LIN {X 0,Y 402.646,Z 650.506,A -85,B 0,C 180,E1 19904.527,E2 19904.527} C_VEL
LIN {X 0,Y 402.658,Z 650.513,A -85,B 0,C 180,E1 19900.591,E2 19900.591} C_VEL
LIN {X 0,Y 402.639,Z 650.511,A -85,B 0,C 180,E1 19896.705,E2 19896.705} C_VEL
LIN {X 0,Y 402.614,Z 650.499,A -85,B 0,C 180,E1 19892.849,E2 19892.849} C_VEL
LIN {X 0,Y 402.66,Z 650.51,A -85,B 0,C 180,E1 19889.006,E2 19889.006} C_VEL
LIN {X 0,Y 402.664,Z 650.497,A -85,B 0,C 180,E1 19885.016,E2 19885.016} C_VEL
LIN {X 0,Y 402.643,Z 650.508,A -85,B 0,C 180,E1 19881.145,E2 19881.145} C_VEL
LIN {X 0,Y 402.604,Z 650.504,A -85,B 0,C 180,E1 19877.232,E2 19877.232} C_VEL
LIN {X 0,Y 402.609,Z 650.515,A -85,B 0,C 180,E1 19873.259,E2 19873.259} C_VEL
LIN {X 0,Y 402.648,Z 650.51,A -85,B 0,C 180,E1 19869.354,E2 19869.354} C_VEL
LIN {X 0,Y 402.661,Z 650.512,A -85,B 0,C 180,E1 19865.502,E2 19865.502} C_VEL
LIN {X 0,Y 402.651,Z 650.512,A -85,B 0,C 180,E1 19861.689,E2 19861.689} C_VEL
LIN {X 0,Y 402.624,Z 650.516,A -85,B 0,C 180,E1 19857.863,E2 19857.863} C_VEL
LIN {X 0,Y 402.648,Z 650.514,A -85,B 0,C 180,E1 19853.95,E2 19853.95} C_VEL
LIN {X 0,Y 402.656,Z 650.511,A -85,B 0,C 180,E1 19851.843,E2 19851.843} C_VEL
LIN {X 0,Y 402.481,Z 651.272,A -85,B 0,C 180,E1 19851.242,E2 19851.242} C_VEL
LIN {X 0,Y 402.023,Z 653.793,A -85,B 0,C 180,E1 19850.558,E2 19850.558} C_VEL
LIN {X 0,Y 401.315,Z 659.057,A -85,B 0,C 180,E1 19849.745,E2 19849.745} C_VEL
LIN {X 0,Y 401.053,Z 668.633,A -85,B 0,C 180,E1 19848.719,E2 19848.719} C_VEL
LIN {X 0,Y 402.027,Z 674.176,A -85,B 0,C 180,E1 19848.104,E2 19848.104} C_VEL
LIN {X 0,Y 409.059,Z 698.473,A -85,B 0,C 180,E1 19845.257,E2 19845.257} C_VEL
LIN {X 0,Y 410.986,Z 706.413,A -85,B 0,C 180,E1 19844.378,E2 19844.378} C_VEL
LIN {X 0,Y 408.514,Z 749.372,A -85,B 0,C 180,E1 19840.433,E2 19840.433} C_VEL
LIN {X 0,Y 406.006,Z 793.704,A -85,B 0,C 180,E1 19836.364,E2 19836.364} C_VEL
LIN {X 0,Y 403.596,Z 838.675,A -85,B 0,C 180,E1 19832.264,E2 19832.264} C_VEL
LIN {X 0,Y 403.179,Z 847.022,A -85,B 0,C 180,E1 19831.548,E2 19831.548} C_VEL
LIN {X 0,Y 399.475,Z 984.558,A -85,B 0,C 180,E1 19828.359,E2 19828.359} C_VEL
LIN {X 0,Y 399.204,Z 1001.716,A -85,B 0,C 180,E1 19827.803,E2 19827.803} C_VEL
LIN {X 0,Y 398.675,Z 1018.522,A -85,B 0,C 180,E1 19826.993,E2 19826.993} C_VEL
LIN {X 0,Y 397.957,Z 1035.489,A -85,B 0,C 180,E1 19825.863,E2 19825.863} C_VEL
LIN {X 0,Y 397.14,Z 1050.63,A -85,B 0,C 180,E1 19824.542,E2 19824.542} C_VEL
LIN {X 0,Y 396.336,Z 1063.911,A -85,B 0,C 180,E1 19823.094,E2 19823.094} C_VEL
LIN {X 0,Y 395.475,Z 1077.222,A -85,B 0,C 180,E1 19821.269,E2 19821.269} C_VEL
LIN {X 0,Y 394.824,Z 1087.41,A -85,B 0,C 180,E1 19819.526,E2 19819.526} C_VEL
LIN {X 0,Y 394.308,Z 1096.659,A -85,B 0,C 180,E1 19817.558,E2 19817.558} C_VEL
LIN {X 0,Y 393.965,Z 1104.345,A -85,B 0,C 180,E1 19815.452,E2 19815.452} C_VEL
LIN {X 0,Y 393.819,Z 1110.47,A -85,B 0,C 180,E1 19813.206,E2 19813.206} C_VEL
LIN {X 0,Y 393.901,Z 1114.817,A -85,B 0,C 180,E1 19810.79,E2 19810.79} C_VEL
LIN {X 0,Y 394.207,Z 1116.994,A -85,B 0,C 180,E1 19808.603,E2 19808.603} C_VEL
LIN {X 0,Y 394.786,Z 1117.402,A -85,B 0,C 180,E1 19806.249,E2 19806.249} C_VEL
LIN {X 0,Y 395.615,Z 1116.078,A -85,B 0,C 180,E1 19804.055,E2 19804.055} C_VEL
LIN {X 0,Y 396.728,Z 1112.949,A -85,B 0,C 180,E1 19801.874,E2 19801.874} C_VEL
LIN {X 0,Y 398.17,Z 1108.026,A -85,B 0,C 180,E1 19799.709,E2 19799.709} C_VEL
LIN {X 0,Y 399.817,Z 1101.607,A -85,B 0,C 180,E1 19797.704,E2 19797.704} C_VEL
LIN {X 0,Y 401.766,Z 1093.191,A -85,B 0,C 180,E1 19795.715,E2 19795.715} C_VEL
LIN {X 0,Y 403.641,Z 1084.014,A -85,B 0,C 180,E1 19794.025,E2 19794.025} C_VEL
LIN {X 0,Y 405.893,Z 1071.581,A -85,B 0,C 180,E1 19792.21,E2 19792.21} C_VEL
LIN {X 0,Y 407.919,Z 1058.287,A -85,B 0,C 180,E1 19790.687,E2 19790.687} C_VEL
LIN {X 0,Y 409.629,Z 1044.619,A -85,B 0,C 180,E1 19789.448,E2 19789.448} C_VEL
LIN {X 0,Y 410.963,Z 1031.006,A -85,B 0,C 180,E1 19788.489,E2 19788.489} C_VEL
LIN {X 0,Y 411.947,Z 1018.129,A -85,B 0,C 180,E1 19787.771,E2 19787.771} C_VEL
LIN {X 0,Y 412.78,Z 1003.186,A -85,B 0,C 180,E1 19787.125,E2 19787.125} C_VEL
LIN {X 0,Y 414.292,Z 966.661,A -85,B 0,C 180,E1 19786.089,E2 19786.089} C_VEL
LIN {X 0,Y 421.684,Z 861.807,A -85,B 0,C 180,E1 19783.324,E2 19783.324} C_VEL
LIN {X 0,Y 426.377,Z 817.793,A -85,B 0,C 180,E1 19779.187,E2 19779.187} C_VEL
LIN {X 0,Y 431.826,Z 773.389,A -85,B 0,C 180,E1 19775,E2 19775} C_VEL
LIN {X 0,Y 437.615,Z 731.795,A -85,B 0,C 180,E1 19771.052,E2 19771.052} C_VEL
LIN {X 0,Y 435.458,Z 721.684,A -85,B 0,C 180,E1 19769.174,E2 19769.174} C_VEL
LIN {X 0,Y 432.981,Z 712.906,A -85,B 0,C 180,E1 19767.13,E2 19767.13} C_VEL
LIN {X 0,Y 430.66,Z 706.333,A -85,B 0,C 180,E1 19765.167,E2 19765.167} C_VEL
LIN {X 0,Y 429.171,Z 702.425,A -85,B 0,C 180,E1 19763.714,E2 19763.714} C_VEL
LIN {X 0,Y 427.98,Z 699.173,A -85,B 0,C 180,E1 19762.255,E2 19762.255} C_VEL
LIN {X 0,Y 426.868,Z 695.743,A -85,B 0,C 180,E1 19760.198,E2 19760.198} C_VEL
LIN {X 0,Y 426.506,Z 695.015,A -85,B 0,C 180,E1 19759.423,E2 19759.423} C_VEL
LIN {X 0,Y 426.307,Z 694.895,A -85,B 0,C 180,E1 19759.043,E2 19759.043} C_VEL
LIN {X 0,Y 424.791,Z 697.509,A -85,B 0,C 180,E1 19758.047,E2 19758.047} C_VEL
LIN {X 0,Y 423.827,Z 699.741,A -85,B 0,C 180,E1 19757.294,E2 19757.294} C_VEL
LIN {X 0,Y 420.94,Z 708.266,A -85,B 0,C 180,E1 19755.654,E2 19755.654} C_VEL
LIN {X 0,Y 437.029,Z 740.937,A -85,B 0,C 180,E1 19753.195,E2 19753.195} C_VEL
LIN {X 0,Y 439.901,Z 747.523,A -85,B 0,C 180,E1 19752.76,E2 19752.76} C_VEL
LIN {X 0,Y 425.069,Z 979.024,A -85,B 0,C 180,E1 19747.665,E2 19747.665} C_VEL
LIN {X 0,Y 422.711,Z 1003.261,A -85,B 0,C 180,E1 19746.883,E2 19746.883} C_VEL
LIN {X 0,Y 419.964,Z 1026.175,A -85,B 0,C 180,E1 19745.884,E2 19745.884} C_VEL
LIN {X 0,Y 417.024,Z 1047.578,A -85,B 0,C 180,E1 19744.7,E2 19744.7} C_VEL
LIN {X 0,Y 413.637,Z 1069.6,A -85,B 0,C 180,E1 19743.201,E2 19743.201} C_VEL
LIN {X 0,Y 410.261,Z 1089.995,A -85,B 0,C 180,E1 19741.516,E2 19741.516} C_VEL
LIN {X 0,Y 406.993,Z 1108.788,A -85,B 0,C 180,E1 19739.67,E2 19739.67} C_VEL
LIN {X 0,Y 403.746,Z 1126.909,A -85,B 0,C 180,E1 19737.547,E2 19737.547} C_VEL
LIN {X 0,Y 400.86,Z 1142.981,A -85,B 0,C 180,E1 19735.324,E2 19735.324} C_VEL
LIN {X 0,Y 398.15,Z 1158.777,A -85,B 0,C 180,E1 19732.75,E2 19732.75} C_VEL
LIN {X 0,Y 396.073,Z 1171.861,A -85,B 0,C 180,E1 19730.232,E2 19730.232} C_VEL
LIN {X 0,Y 394.432,Z 1183.554,A -85,B 0,C 180,E1 19727.555,E2 19727.555} C_VEL
LIN {X 0,Y 393.294,Z 1193.275,A -85,B 0,C 180,E1 19724.877,E2 19724.877} C_VEL
LIN {X 0,Y 392.561,Z 1201.854,A -85,B 0,C 180,E1 19722.009,E2 19722.009} C_VEL
LIN {X 0,Y 392.233,Z 1208.397,A -85,B 0,C 180,E1 19719.24,E2 19719.24} C_VEL
LIN {X 0,Y 392.151,Z 1213.369,A -85,B 0,C 180,E1 19716.439,E2 19716.439} C_VEL
LIN {X 0,Y 392.187,Z 1216.843,A -85,B 0,C 180,E1 19713.652,E2 19713.652} C_VEL
LIN {X 0,Y 392.216,Z 1218.667,A -85,B 0,C 180,E1 19710.874,E2 19710.874} C_VEL
LIN {X 0,Y 392.161,Z 1219.127,A -85,B 0,C 180,E1 19708.099,E2 19708.099} C_VEL
LIN {X 0,Y 392.064,Z 1217.981,A -85,B 0,C 180,E1 19705.317,E2 19705.317} C_VEL
LIN {X 0,Y 392.055,Z 1215.324,A -85,B 0,C 180,E1 19702.377,E2 19702.377} C_VEL
LIN {X 0,Y 392.305,Z 1211.002,A -85,B 0,C 180,E1 19699.424,E2 19699.424} C_VEL
LIN {X 0,Y 393.041,Z 1204.73,A -85,B 0,C 180,E1 19696.313,E2 19696.313} C_VEL
LIN {X 0,Y 394.347,Z 1197.092,A -85,B 0,C 180,E1 19693.349,E2 19693.349} C_VEL
LIN {X 0,Y 396.474,Z 1187.039,A -85,B 0,C 180,E1 19690.247,E2 19690.247} C_VEL
LIN {X 0,Y 399.332,Z 1175.533,A -85,B 0,C 180,E1 19687.317,E2 19687.317} C_VEL
LIN {X 0,Y 403.067,Z 1161.949,A -85,B 0,C 180,E1 19684.427,E2 19684.427} C_VEL
LIN {X 0,Y 407.523,Z 1146.959,A -85,B 0,C 180,E1 19681.734,E2 19681.734} C_VEL
LIN {X 0,Y 413.055,Z 1129.099,A -85,B 0,C 180,E1 19679.041,E2 19679.041} C_VEL
LIN {X 0,Y 419.266,Z 1109.523,A -85,B 0,C 180,E1 19676.569,E2 19676.569} C_VEL
LIN {X 0,Y 425.881,Z 1088.959,A -85,B 0,C 180,E1 19674.389,E2 19674.389} C_VEL
LIN {X 0,Y 433,Z 1066.974,A -85,B 0,C 180,E1 19672.436,E2 19672.436} C_VEL
LIN {X 0,Y 440.578,Z 1043.466,A -85,B 0,C 180,E1 19670.713,E2 19670.713} C_VEL
LIN {X 0,Y 448.214,Z 1019.183,A -85,B 0,C 180,E1 19669.267,E2 19669.267} C_VEL
LIN {X 0,Y 455.498,Z 995.065,A -85,B 0,C 180,E1 19668.137,E2 19668.137} C_VEL
LIN {X 0,Y 462.97,Z 967.876,A -85,B 0,C 180,E1 19667.141,E2 19667.141} C_VEL
LIN {X 0,Y 483.825,Z 882.658,A -85,B 0,C 180,E1 19664.617,E2 19664.617} C_VEL
LIN {X 0,Y 466.018,Z 953.723,A -85,B 0,C 180,E1 19662.524,E2 19662.524} C_VEL
LIN {X 0,Y 459.927,Z 976.756,A -85,B 0,C 180,E1 19661.621,E2 19661.621} C_VEL
LIN {X 0,Y 453.131,Z 999.954,A -85,B 0,C 180,E1 19660.45,E2 19660.45} C_VEL
LIN {X 0,Y 446.12,Z 1022.308,A -85,B 0,C 180,E1 19659.038,E2 19659.038} C_VEL
LIN {X 0,Y 438.753,Z 1044.675,A -85,B 0,C 180,E1 19657.31,E2 19657.31} C_VEL
LIN {X 0,Y 431.735,Z 1065.276,A -85,B 0,C 180,E1 19655.383,E2 19655.383} C_VEL
LIN {X 0,Y 425.061,Z 1084.433,A -85,B 0,C 180,E1 19653.239,E2 19653.239} C_VEL
LIN {X 0,Y 418.789,Z 1102.064,A -85,B 0,C 180,E1 19650.889,E2 19650.889} C_VEL
LIN {X 0,Y 413.031,Z 1118.126,A -85,B 0,C 180,E1 19648.329,E2 19648.329} C_VEL
LIN {X 0,Y 408.086,Z 1131.941,A -85,B 0,C 180,E1 19645.704,E2 19645.704} C_VEL
LIN {X 0,Y 403.945,Z 1143.775,A -85,B 0,C 180,E1 19643.026,E2 19643.026} C_VEL
LIN {X 0,Y 400.198,Z 1154.642,A -85,B 0,C 180,E1 19640.019,E2 19640.019} C_VEL
LIN {X 0,Y 397.338,Z 1163.443,A -85,B 0,C 180,E1 19637.005,E2 19637.005} C_VEL
LIN {X 0,Y 395.122,Z 1170.858,A -85,B 0,C 180,E1 19633.764,E2 19633.764} C_VEL
LIN {X 0,Y 393.737,Z 1176.111,A -85,B 0,C 180,E1 19630.686,E2 19630.686} C_VEL
LIN {X 0,Y 392.874,Z 1179.647,A -85,B 0,C 180,E1 19627.608,E2 19627.608} C_VEL
LIN {X 0,Y 392.42,Z 1181.535,A -85,B 0,C 180,E1 19624.533,E2 19624.533} C_VEL
LIN {X 0,Y 392.235,Z 1181.899,A -85,B 0,C 180,E1 19621.61,E2 19621.61} C_VEL
LIN {X 0,Y 392.162,Z 1180.769,A -85,B 0,C 180,E1 19618.834,E2 19618.834} C_VEL
LIN {X 0,Y 392.176,Z 1177.983,A -85,B 0,C 180,E1 19615.763,E2 19615.763} C_VEL
LIN {X 0,Y 392.357,Z 1173.769,A -85,B 0,C 180,E1 19612.83,E2 19612.83} C_VEL
LIN {X 0,Y 392.769,Z 1167.777,A -85,B 0,C 180,E1 19609.887,E2 19609.887} C_VEL
LIN {X 0,Y 393.54,Z 1160.062,A -85,B 0,C 180,E1 19606.934,E2 19606.934} C_VEL
LIN {X 0,Y 394.697,Z 1150.979,A -85,B 0,C 180,E1 19604.125,E2 19604.125} C_VEL
LIN {X 0,Y 396.355,Z 1139.874,A -85,B 0,C 180,E1 19601.318,E2 19601.318} C_VEL
LIN {X 0,Y 398.437,Z 1127.317,A -85,B 0,C 180,E1 19598.665,E2 19598.665} C_VEL
LIN {X 0,Y 401.054,Z 1112.484,A -85,B 0,C 180,E1 19596.026,E2 19596.026} C_VEL
LIN {X 0,Y 403.937,Z 1096.683,A -85,B 0,C 180,E1 19593.65,E2 19593.65} C_VEL
LIN {X 0,Y 407.051,Z 1079.568,A -85,B 0,C 180,E1 19591.464,E2 19591.464} C_VEL
LIN {X 0,Y 410.306,Z 1060.961,A -85,B 0,C 180,E1 19589.467,E2 19589.467} C_VEL
LIN {X 0,Y 413.532,Z 1041.496,A -85,B 0,C 180,E1 19587.704,E2 19587.704} C_VEL
LIN {X 0,Y 416.755,Z 1020.503,A -85,B 0,C 180,E1 19586.114,E2 19586.114} C_VEL
LIN {X 0,Y 419.661,Z 999.367,A -85,B 0,C 180,E1 19584.793,E2 19584.793} C_VEL
LIN {X 0,Y 422.338,Z 977.144,A -85,B 0,C 180,E1 19583.672,E2 19583.672} C_VEL
LIN {X 0,Y 424.639,Z 953.609,A -85,B 0,C 180,E1 19582.759,E2 19582.759} C_VEL
LIN {X 0,Y 426.356,Z 930.684,A -85,B 0,C 180,E1 19582.109,E2 19582.109} C_VEL
LIN {X 0,Y 438.997,Z 728.954,A -85,B 0,C 180,E1 19577.705,E2 19577.705} C_VEL
LIN {X 0,Y 420.147,Z 695.163,A -85,B 0,C 180,E1 19574.978,E2 19574.978} C_VEL
LIN {X 0,Y 403.964,Z 667.893,A -85,B 0,C 180,E1 19572.44,E2 19572.44} C_VEL
LIN {X 0,Y 396.718,Z 655.938,A -85,B 0,C 180,E1 19571.232,E2 19571.232} C_VEL
LIN {X 0,Y 394.919,Z 652.752,A -85,B 0,C 180,E1 19570.918,E2 19570.918} C_VEL
LIN {X 0,Y 394.665,Z 651.506,A -85,B 0,C 180,E1 19570.819,E2 19570.819} C_VEL
LIN {X 0,Y 394.674,Z 651.506,A -85,B 0,C 180,E1 19566.822,E2 19566.822} C_VEL
LIN {X 0,Y 394.713,Z 651.496,A -85,B 0,C 180,E1 19562.829,E2 19562.829} C_VEL
LIN {X 0,Y 394.726,Z 651.495,A -85,B 0,C 180,E1 19558.937,E2 19558.937} C_VEL
LIN {X 0,Y 394.696,Z 651.503,A -85,B 0,C 180,E1 19555.03,E2 19555.03} C_VEL
LIN {X 0,Y 394.665,Z 651.508,A -85,B 0,C 180,E1 19551.087,E2 19551.087} C_VEL
LIN {X 0,Y 394.702,Z 651.497,A -85,B 0,C 180,E1 19547.243,E2 19547.243} C_VEL
LIN {X 0,Y 394.727,Z 651.485,A -85,B 0,C 180,E1 19543.329,E2 19543.329} C_VEL
LIN {X 0,Y 394.719,Z 651.492,A -85,B 0,C 180,E1 19539.332,E2 19539.332} C_VEL
LIN {X 0,Y 394.688,Z 651.505,A -85,B 0,C 180,E1 19535.415,E2 19535.415} C_VEL
LIN {X 0,Y 394.694,Z 651.492,A -85,B 0,C 180,E1 19531.308,E2 19531.308} C_VEL
LIN {X 0,Y 394.72,Z 651.487,A -85,B 0,C 180,E1 19527.389,E2 19527.389} C_VEL
LIN {X 0,Y 394.715,Z 651.5,A -85,B 0,C 180,E1 19523.457,E2 19523.457} C_VEL
LIN {X 0,Y 394.682,Z 651.483,A -85,B 0,C 180,E1 19519.492,E2 19519.492} C_VEL
LIN {X 0,Y 394.649,Z 651.506,A -85,B 0,C 180,E1 19515.476,E2 19515.476} C_VEL
LIN {X 0,Y 394.684,Z 651.503,A -85,B 0,C 180,E1 19511.541,E2 19511.541} C_VEL
LIN {X 0,Y 394.717,Z 651.502,A -85,B 0,C 180,E1 19507.599,E2 19507.599} C_VEL
LIN {X 0,Y 394.724,Z 651.498,A -85,B 0,C 180,E1 19503.688,E2 19503.688} C_VEL
LIN {X 0,Y 394.692,Z 651.504,A -85,B 0,C 180,E1 19499.745,E2 19499.745} C_VEL
LIN {X 0,Y 394.687,Z 651.506,A -85,B 0,C 180,E1 19495.781,E2 19495.781} C_VEL
LIN {X 0,Y 394.717,Z 651.5,A -85,B 0,C 180,E1 19491.826,E2 19491.826} C_VEL
LIN {X 0,Y 394.735,Z 651.678,A -85,B 0,C 180,E1 19490.866,E2 19490.866} C_VEL
LIN {X 0,Y 402.027,Z 674.176,A -85,B 0,C 180,E1 19488.104,E2 19488.104} C_VEL
LIN {X 0,Y 402.871,Z 680.333,A -85,B 0,C 180,E1 19487.442,E2 19487.442} C_VEL
LIN {X 0,Y 401.632,Z 699.052,A -85,B 0,C 180,E1 19485.691,E2 19485.691} C_VEL
LIN {X 0,Y 402.317,Z 703.478,A -85,B 0,C 180,E1 19485.217,E2 19485.217} C_VEL
LIN {X 0,Y 403.454,Z 708.427,A -85,B 0,C 180,E1 19484.665,E2 19484.665} C_VEL
LIN {X 0,Y 400.84,Z 752.044,A -85,B 0,C 180,E1 19480.616,E2 19480.616} C_VEL
LIN {X 0,Y 398.274,Z 796.537,A -85,B 0,C 180,E1 19476.508,E2 19476.508} C_VEL
LIN {X 0,Y 395.755,Z 842.489,A -85,B 0,C 180,E1 19472.272,E2 19472.272} C_VEL
LIN {X 0,Y 395.417,Z 847.822,A -85,B 0,C 180,E1 19471.823,E2 19471.823} C_VEL
LIN {X 0,Y 391.587,Z 985.022,A -85,B 0,C 180,E1 19468.547,E2 19468.547} C_VEL
LIN {X 0,Y 391.307,Z 1002.317,A -85,B 0,C 180,E1 19467.979,E2 19467.979} C_VEL
LIN {X 0,Y 390.777,Z 1018.864,A -85,B 0,C 180,E1 19467.172,E2 19467.172} C_VEL
LIN {X 0,Y 390.074,Z 1035.219,A -85,B 0,C 180,E1 19466.075,E2 19466.075} C_VEL
LIN {X 0,Y 389.296,Z 1049.667,A -85,B 0,C 180,E1 19464.827,E2 19464.827} C_VEL
LIN {X 0,Y 388.394,Z 1064.416,A -85,B 0,C 180,E1 19463.217,E2 19463.217} C_VEL
LIN {X 0,Y 387.569,Z 1076.966,A -85,B 0,C 180,E1 19461.487,E2 19461.487} C_VEL
LIN {X 0,Y 386.868,Z 1087.854,A -85,B 0,C 180,E1 19459.629,E2 19459.629} C_VEL
LIN {X 0,Y 386.309,Z 1097.863,A -85,B 0,C 180,E1 19457.469,E2 19457.469} C_VEL
LIN {X 0,Y 385.974,Z 1105.522,A -85,B 0,C 180,E1 19455.318,E2 19455.318} C_VEL
LIN {X 0,Y 385.846,Z 1111.603,A -85,B 0,C 180,E1 19453.026,E2 19453.026} C_VEL
LIN {X 0,Y 385.959,Z 1115.863,A -85,B 0,C 180,E1 19450.596,E2 19450.596} C_VEL
LIN {X 0,Y 386.312,Z 1118.066,A -85,B 0,C 180,E1 19448.331,E2 19448.331} C_VEL
LIN {X 0,Y 386.959,Z 1118.458,A -85,B 0,C 180,E1 19445.929,E2 19445.929} C_VEL
LIN {X 0,Y 387.871,Z 1117.094,A -85,B 0,C 180,E1 19443.692,E2 19443.692} C_VEL
LIN {X 0,Y 389.181,Z 1113.683,A -85,B 0,C 180,E1 19441.322,E2 19441.322} C_VEL
LIN {X 0,Y 390.768,Z 1108.625,A -85,B 0,C 180,E1 19439.117,E2 19439.117} C_VEL
LIN {X 0,Y 392.704,Z 1101.473,A -85,B 0,C 180,E1 19436.932,E2 19436.932} C_VEL
LIN {X 0,Y 394.668,Z 1093.37,A -85,B 0,C 180,E1 19435.055,E2 19435.055} C_VEL
LIN {X 0,Y 396.877,Z 1083.175,A -85,B 0,C 180,E1 19433.197,E2 19433.197} C_VEL
LIN {X 0,Y 399.022,Z 1071.886,A -85,B 0,C 180,E1 19431.568,E2 19431.568} C_VEL
LIN {X 0,Y 401.176,Z 1058.387,A -85,B 0,C 180,E1 19430.022,E2 19430.022} C_VEL
LIN {X 0,Y 403.1,Z 1043.582,A -85,B 0,C 180,E1 19428.696,E2 19428.696} C_VEL
LIN {X 0,Y 404.436,Z 1030.633,A -85,B 0,C 180,E1 19427.794,E2 19427.794} C_VEL
LIN {X 0,Y 405.446,Z 1018.234,A -85,B 0,C 180,E1 19427.101,E2 19427.101} C_VEL
LIN {X 0,Y 406.28,Z 1003.609,A -85,B 0,C 180,E1 19426.472,E2 19426.472} C_VEL
LIN {X 0,Y 408.076,Z 964.911,A -85,B 0,C 180,E1 19425.356,E2 19425.356} C_VEL
LIN {X 0,Y 415.65,Z 863.65,A -85,B 0,C 180,E1 19422.642,E2 19422.642} C_VEL
LIN {X 0,Y 420.636,Z 820.445,A -85,B 0,C 180,E1 19418.524,E2 19418.524} C_VEL
LIN {X 0,Y 426.779,Z 774.226,A -85,B 0,C 180,E1 19414.108,E2 19414.108} C_VEL
LIN {X 0,Y 432.533,Z 736.055,A -85,B 0,C 180,E1 19410.416,E2 19410.416} C_VEL
LIN {X 0,Y 430.698,Z 726.646,A -85,B 0,C 180,E1 19408.585,E2 19408.585} C_VEL
LIN {X 0,Y 428.479,Z 718.439,A -85,B 0,C 180,E1 19406.581,E2 19406.581} C_VEL
LIN {X 0,Y 426.54,Z 712.406,A -85,B 0,C 180,E1 19404.66,E2 19404.66} C_VEL
LIN {X 0,Y 425.512,Z 709.318,A -85,B 0,C 180,E1 19403.475,E2 19403.475} C_VEL
LIN {X 0,Y 424.538,Z 706.275,A -85,B 0,C 180,E1 19402.066,E2 19402.066} C_VEL
LIN {X 0,Y 423.625,Z 703.028,A -85,B 0,C 180,E1 19400.056,E2 19400.056} C_VEL
LIN {X 0,Y 423.337,Z 702.308,A -85,B 0,C 180,E1 19399.248,E2 19399.248} C_VEL
LIN {X 0,Y 421.274,Z 706.106,A -85,B 0,C 180,E1 19397.874,E2 19397.874} C_VEL
LIN {X 0,Y 417.335,Z 717.08,A -85,B 0,C 180,E1 19395.741,E2 19395.741} C_VEL
LIN {X 0,Y 433.11,Z 749.566,A -85,B 0,C 180,E1 19393.301,E2 19393.301} C_VEL
LIN {X 0,Y 417.912,Z 978.657,A -85,B 0,C 180,E1 19388.153,E2 19388.153} C_VEL
LIN {X 0,Y 415.516,Z 1002.68,A -85,B 0,C 180,E1 19387.364,E2 19387.364} C_VEL
LIN {X 0,Y 412.727,Z 1025.325,A -85,B 0,C 180,E1 19386.363,E2 19386.363} C_VEL
LIN {X 0,Y 409.688,Z 1046.975,A -85,B 0,C 180,E1 19385.151,E2 19385.151} C_VEL
LIN {X 0,Y 406.211,Z 1069.033,A -85,B 0,C 180,E1 19383.628,E2 19383.628} C_VEL
LIN {X 0,Y 402.754,Z 1089.393,A -85,B 0,C 180,E1 19381.922,E2 19381.922} C_VEL
LIN {X 0,Y 399.402,Z 1108.229,A -85,B 0,C 180,E1 19380.043,E2 19380.043} C_VEL
LIN {X 0,Y 396.006,Z 1126.687,A -85,B 0,C 180,E1 19377.844,E2 19377.844} C_VEL
LIN {X 0,Y 393.005,Z 1142.992,A -85,B 0,C 180,E1 19375.544,E2 19375.544} C_VEL
LIN {X 0,Y 390.378,Z 1157.917,A -85,B 0,C 180,E1 19373.069,E2 19373.069} C_VEL
LIN {X 0,Y 388.226,Z 1171.099,A -85,B 0,C 180,E1 19370.501,E2 19370.501} C_VEL
LIN {X 0,Y 386.523,Z 1182.843,A -85,B 0,C 180,E1 19367.771,E2 19367.771} C_VEL
LIN {X 0,Y 385.344,Z 1192.641,A -85,B 0,C 180,E1 19365.037,E2 19365.037} C_VEL
LIN {X 0,Y 384.594,Z 1201.167,A -85,B 0,C 180,E1 19362.155,E2 19362.155} C_VEL
LIN {X 0,Y 384.249,Z 1207.849,A -85,B 0,C 180,E1 19359.282,E2 19359.282} C_VEL
LIN {X 0,Y 384.168,Z 1212.862,A -85,B 0,C 180,E1 19356.424,E2 19356.424} C_VEL
LIN {X 0,Y 384.206,Z 1216.352,A -85,B 0,C 180,E1 19353.579,E2 19353.579} C_VEL
LIN {X 0,Y 384.231,Z 1218.201,A -85,B 0,C 180,E1 19350.743,E2 19350.743} C_VEL
LIN {X 0,Y 384.167,Z 1218.671,A -85,B 0,C 180,E1 19347.91,E2 19347.91} C_VEL
LIN {X 0,Y 384.061,Z 1217.536,A -85,B 0,C 180,E1 19345.069,E2 19345.069} C_VEL
LIN {X 0,Y 384.063,Z 1214.9,A -85,B 0,C 180,E1 19342.067,E2 19342.067} C_VEL
LIN {X 0,Y 384.366,Z 1210.584,A -85,B 0,C 180,E1 19339.051,E2 19339.051} C_VEL
LIN {X 0,Y 385.255,Z 1204.012,A -85,B 0,C 180,E1 19335.724,E2 19335.724} C_VEL
LIN {X 0,Y 386.824,Z 1195.882,A -85,B 0,C 180,E1 19332.55,E2 19332.55} C_VEL
LIN {X 0,Y 389.23,Z 1185.771,A -85,B 0,C 180,E1 19329.392,E2 19329.392} C_VEL
LIN {X 0,Y 392.405,Z 1174.164,A -85,B 0,C 180,E1 19326.417,E2 19326.417} C_VEL
LIN {X 0,Y 396.748,Z 1159.803,A -85,B 0,C 180,E1 19323.345,E2 19323.345} C_VEL
LIN {X 0,Y 401.919,Z 1143.803,A -85,B 0,C 180,E1 19320.488,E2 19320.488} C_VEL
LIN {X 0,Y 407.83,Z 1126.286,A -85,B 0,C 180,E1 19317.856,E2 19317.856} C_VEL
LIN {X 0,Y 414.605,Z 1106.761,A -85,B 0,C 180,E1 19315.391,E2 19315.391} C_VEL
LIN {X 0,Y 421.996,Z 1085.741,A -85,B 0,C 180,E1 19313.167,E2 19313.167} C_VEL
LIN {X 0,Y 429.966,Z 1063.264,A -85,B 0,C 180,E1 19311.19,E2 19311.19} C_VEL
LIN {X 0,Y 438.413,Z 1039.238,A -85,B 0,C 180,E1 19309.457,E2 19309.457} C_VEL
LIN {X 0,Y 446.678,Z 1015.23,A -85,B 0,C 180,E1 19308.071,E2 19308.071} C_VEL
LIN {X 0,Y 454.455,Z 991.415,A -85,B 0,C 180,E1 19306.994,E2 19306.994} C_VEL
LIN {X 0,Y 462.394,Z 964.567,A -85,B 0,C 180,E1 19306.04,E2 19306.04} C_VEL
LIN {X 0,Y 474.662,Z 916.991,A -85,B 0,C 180,E1 19304.622,E2 19304.622} C_VEL
LIN {X 0,Y 463.429,Z 959.702,A -85,B 0,C 180,E1 19303.326,E2 19303.326} C_VEL
LIN {X 0,Y 456.454,Z 983.213,A -85,B 0,C 180,E1 19302.348,E2 19302.348} C_VEL
LIN {X 0,Y 448.781,Z 1006.559,A -85,B 0,C 180,E1 19301.094,E2 19301.094} C_VEL
LIN {X 0,Y 440.915,Z 1028.975,A -85,B 0,C 180,E1 19299.589,E2 19299.589} C_VEL
LIN {X 0,Y 433.026,Z 1050.608,A -85,B 0,C 180,E1 19297.814,E2 19297.814} C_VEL
LIN {X 0,Y 425.278,Z 1071.277,A -85,B 0,C 180,E1 19295.753,E2 19295.753} C_VEL
LIN {X 0,Y 418.168,Z 1089.948,A -85,B 0,C 180,E1 19293.531,E2 19293.531} C_VEL
LIN {X 0,Y 411.364,Z 1107.559,A -85,B 0,C 180,E1 19291.02,E2 19291.02} C_VEL
LIN {X 0,Y 405.16,Z 1123.521,A -85,B 0,C 180,E1 19288.286,E2 19288.286} C_VEL
LIN {X 0,Y 399.882,Z 1137.117,A -85,B 0,C 180,E1 19285.475,E2 19285.475} C_VEL
LIN {X 0,Y 395.49,Z 1148.605,A -85,B 0,C 180,E1 19282.603,E2 19282.603} C_VEL
LIN {X 0,Y 391.798,Z 1158.672,A -85,B 0,C 180,E1 19279.534,E2 19279.534} C_VEL
LIN {X 0,Y 388.975,Z 1166.853,A -85,B 0,C 180,E1 19276.428,E2 19276.428} C_VEL
LIN {X 0,Y 386.955,Z 1173.258,A -85,B 0,C 180,E1 19273.299,E2 19273.299} C_VEL
LIN {X 0,Y 385.591,Z 1177.858,A -85,B 0,C 180,E1 19270.159,E2 19270.159} C_VEL
LIN {X 0,Y 384.765,Z 1180.975,A -85,B 0,C 180,E1 19266.869,E2 19266.869} C_VEL
LIN {X 0,Y 384.386,Z 1182.339,A -85,B 0,C 180,E1 19263.881,E2 19263.881} C_VEL
LIN {X 0,Y 384.217,Z 1182.094,A -85,B 0,C 180,E1 19260.898,E2 19260.898} C_VEL
LIN {X 0,Y 384.155,Z 1180.301,A -85,B 0,C 180,E1 19257.766,E2 19257.766} C_VEL
LIN {X 0,Y 384.219,Z 1177.239,A -85,B 0,C 180,E1 19254.927,E2 19254.927} C_VEL
LIN {X 0,Y 384.456,Z 1172.39,A -85,B 0,C 180,E1 19251.93,E2 19251.93} C_VEL
LIN {X 0,Y 384.981,Z 1165.902,A -85,B 0,C 180,E1 19248.923,E2 19248.923} C_VEL
LIN {X 0,Y 385.905,Z 1157.583,A -85,B 0,C 180,E1 19245.907,E2 19245.907} C_VEL
LIN {X 0,Y 387.256,Z 1147.73,A -85,B 0,C 180,E1 19243.04,E2 19243.04} C_VEL
LIN {X 0,Y 389.145,Z 1135.888,A -85,B 0,C 180,E1 19240.178,E2 19240.178} C_VEL
LIN {X 0,Y 391.34,Z 1123.384,A -85,B 0,C 180,E1 19237.627,E2 19237.627} C_VEL
LIN {X 0,Y 394.043,Z 1108.674,A -85,B 0,C 180,E1 19235.092,E2 19235.092} C_VEL
LIN {X 0,Y 397.025,Z 1092.604,A -85,B 0,C 180,E1 19232.752,E2 19232.752} C_VEL
LIN {X 0,Y 400.345,Z 1074.618,A -85,B 0,C 180,E1 19230.531,E2 19230.531} C_VEL
LIN {X 0,Y 403.803,Z 1055.148,A -85,B 0,C 180,E1 19228.506,E2 19228.506} C_VEL
LIN {X 0,Y 407.073,Z 1035.559,A -85,B 0,C 180,E1 19226.791,E2 19226.791} C_VEL
LIN {X 0,Y 410.344,Z 1014.252,A -85,B 0,C 180,E1 19225.241,E2 19225.241} C_VEL
LIN {X 0,Y 413.297,Z 992.366,A -85,B 0,C 180,E1 19223.95,E2 19223.95} C_VEL
LIN {X 0,Y 415.883,Z 969.815,A -85,B 0,C 180,E1 19222.886,E2 19222.886} C_VEL
LIN {X 0,Y 418.114,Z 945.816,A -85,B 0,C 180,E1 19222.022,E2 19222.022} C_VEL
LIN {X 0,Y 420.091,Z 917.398,A -85,B 0,C 180,E1 19221.306,E2 19221.306} C_VEL
LIN {X 0,Y 432.144,Z 731.726,A -85,B 0,C 180,E1 19217.18,E2 19217.18} C_VEL
LIN {X 0,Y 413.501,Z 698.183,A -85,B 0,C 180,E1 19214.408,E2 19214.408} C_VEL
LIN {X 0,Y 396.406,Z 669.438,A -85,B 0,C 180,E1 19211.657,E2 19211.657} C_VEL
LIN {X 0,Y 389.378,Z 657.671,A -85,B 0,C 180,E1 19210.447,E2 19210.447} C_VEL
LIN {X 0,Y 387.126,Z 654.072,A -85,B 0,C 180,E1 19210.052,E2 19210.052} C_VEL
LIN {X 0,Y 386.751,Z 652.489,A -85,B 0,C 180,E1 19209.933,E2 19209.933} C_VEL
LIN {X 0,Y 386.77,Z 652.487,A -85,B 0,C 180,E1 19205.935,E2 19205.935} C_VEL
LIN {X 0,Y 386.789,Z 652.483,A -85,B 0,C 180,E1 19202.004,E2 19202.004} C_VEL
LIN {X 0,Y 386.779,Z 652.493,A -85,B 0,C 180,E1 19198.069,E2 19198.069} C_VEL
LIN {X 0,Y 386.746,Z 652.497,A -85,B 0,C 180,E1 19194.112,E2 19194.112} C_VEL
LIN {X 0,Y 386.73,Z 652.499,A -85,B 0,C 180,E1 19190.115,E2 19190.115} C_VEL
LIN {X 0,Y 386.768,Z 652.491,A -85,B 0,C 180,E1 19186.215,E2 19186.215} C_VEL
LIN {X 0,Y 386.781,Z 652.483,A -85,B 0,C 180,E1 19182.24,E2 19182.24} C_VEL
LIN {X 0,Y 386.751,Z 652.478,A -85,B 0,C 180,E1 19178.177,E2 19178.177} C_VEL
LIN {X 0,Y 386.712,Z 652.492,A -85,B 0,C 180,E1 19174.154,E2 19174.154} C_VEL
LIN {X 0,Y 386.737,Z 652.492,A -85,B 0,C 180,E1 19170.002,E2 19170.002} C_VEL
LIN {X 0,Y 386.771,Z 652.468,A -85,B 0,C 180,E1 19166,E2 19166} C_VEL
LIN {X 0,Y 386.78,Z 652.489,A -85,B 0,C 180,E1 19161.978,E2 19161.978} C_VEL
LIN {X 0,Y 386.742,Z 652.47,A -85,B 0,C 180,E1 19158.065,E2 19158.065} C_VEL
LIN {X 0,Y 386.732,Z 652.492,A -85,B 0,C 180,E1 19154.096,E2 19154.096} C_VEL
LIN {X 0,Y 386.77,Z 652.486,A -85,B 0,C 180,E1 19150.207,E2 19150.207} C_VEL
LIN {X 0,Y 386.789,Z 652.484,A -85,B 0,C 180,E1 19146.213,E2 19146.213} C_VEL
LIN {X 0,Y 386.792,Z 652.488,A -85,B 0,C 180,E1 19142.105,E2 19142.105} C_VEL
LIN {X 0,Y 386.756,Z 652.493,A -85,B 0,C 180,E1 19138.173,E2 19138.173} C_VEL
LIN {X 0,Y 386.772,Z 652.492,A -85,B 0,C 180,E1 19134.008,E2 19134.008} C_VEL
LIN {X 0,Y 386.798,Z 652.736,A -85,B 0,C 180,E1 19131.373,E2 19131.373} C_VEL
LIN {X 0,Y 395.161,Z 678.424,A -85,B 0,C 180,E1 19128.187,E2 19128.187} C_VEL
LIN {X 0,Y 402.03,Z 702.438,A -85,B 0,C 180,E1 19125.336,E2 19125.336} C_VEL
LIN {X 0,Y 402.317,Z 703.478,A -85,B 0,C 180,E1 19125.217,E2 19125.217} C_VEL
LIN {X 0,Y 402.255,Z 707.115,A -85,B 0,C 180,E1 19124.872,E2 19124.872} C_VEL
LIN {X 0,Y 399.861,Z 712.81,A -85,B 0,C 180,E1 19124.481,E2 19124.481} C_VEL
LIN {X 0,Y 395.849,Z 720.554,A -85,B 0,C 180,E1 19123.985,E2 19123.985} C_VEL
LIN {X 0,Y 395.104,Z 723.822,A -85,B 0,C 180,E1 19123.709,E2 19123.709} C_VEL
LIN {X 0,Y 392.431,Z 767.034,A -85,B 0,C 180,E1 19119.657,E2 19119.657} C_VEL
LIN {X 0,Y 389.812,Z 810.492,A -85,B 0,C 180,E1 19115.603,E2 19115.603} C_VEL
LIN {X 0,Y 387.669,Z 848.21,A -85,B 0,C 180,E1 19112.112,E2 19112.112} C_VEL
LIN {X 0,Y 383.707,Z 985.121,A -85,B 0,C 180,E1 19108.751,E2 19108.751} C_VEL
LIN {X 0,Y 383.42,Z 1002.699,A -85,B 0,C 180,E1 19108.17,E2 19108.17} C_VEL
LIN {X 0,Y 382.882,Z 1019.167,A -85,B 0,C 180,E1 19107.358,E2 19107.358} C_VEL
LIN {X 0,Y 382.211,Z 1034.656,A -85,B 0,C 180,E1 19106.318,E2 19106.318} C_VEL
LIN {X 0,Y 381.412,Z 1049.478,A -85,B 0,C 180,E1 19105.044,E2 19105.044} C_VEL
LIN {X 0,Y 380.515,Z 1063.892,A -85,B 0,C 180,E1 19103.467,E2 19103.467} C_VEL
LIN {X 0,Y 379.704,Z 1076.198,A -85,B 0,C 180,E1 19101.792,E2 19101.792} C_VEL
LIN {X 0,Y 378.964,Z 1087.433,A -85,B 0,C 180,E1 19099.895,E2 19099.895} C_VEL
LIN {X 0,Y 378.4,Z 1097.074,A -85,B 0,C 180,E1 19097.846,E2 19097.846} C_VEL
LIN {X 0,Y 378.033,Z 1105.206,A -85,B 0,C 180,E1 19095.648,E2 19095.648} C_VEL
LIN {X 0,Y 377.874,Z 1111.263,A -85,B 0,C 180,E1 19093.462,E2 19093.462} C_VEL
LIN {X 0,Y 377.973,Z 1116.321,A -85,B 0,C 180,E1 19090.822,E2 19090.822} C_VEL
LIN {X 0,Y 378.355,Z 1118.947,A -85,B 0,C 180,E1 19088.354,E2 19088.354} C_VEL
LIN {X 0,Y 379.006,Z 1119.586,A -85,B 0,C 180,E1 19085.987,E2 19085.987} C_VEL
LIN {X 0,Y 379.992,Z 1118.416,A -85,B 0,C 180,E1 19083.617,E2 19083.617} C_VEL
LIN {X 0,Y 381.278,Z 1115.526,A -85,B 0,C 180,E1 19081.349,E2 19081.349} C_VEL
LIN {X 0,Y 383.038,Z 1110.41,A -85,B 0,C 180,E1 19078.95,E2 19078.95} C_VEL
LIN {X 0,Y 384.927,Z 1104.061,A -85,B 0,C 180,E1 19076.87,E2 19076.87} C_VEL
LIN {X 0,Y 387.148,Z 1095.752,A -85,B 0,C 180,E1 19074.811,E2 19074.811} C_VEL
LIN {X 0,Y 389.463,Z 1085.856,A -85,B 0,C 180,E1 19072.918,E2 19072.918} C_VEL
LIN {X 0,Y 391.81,Z 1074.401,A -85,B 0,C 180,E1 19071.189,E2 19071.189} C_VEL
LIN {X 0,Y 394.1,Z 1061.332,A -85,B 0,C 180,E1 19069.619,E2 19069.619} C_VEL
LIN {X 0,Y 396.046,Z 1048.007,A -85,B 0,C 180,E1 19068.345,E2 19068.345} C_VEL
LIN {X 0,Y 397.673,Z 1033.75,A -85,B 0,C 180,E1 19067.288,E2 19067.288} C_VEL
LIN {X 0,Y 398.847,Z 1020.461,A -85,B 0,C 180,E1 19066.515,E2 19066.515} C_VEL
LIN {X 0,Y 399.83,Z 1005.164,A -85,B 0,C 180,E1 19065.829,E2 19065.829} C_VEL
LIN {X 0,Y 401.71,Z 967.98,A -85,B 0,C 180,E1 19064.713,E2 19064.713} C_VEL
LIN {X 0,Y 409.816,Z 864.936,A -85,B 0,C 180,E1 19061.873,E2 19061.873} C_VEL
LIN {X 0,Y 415.448,Z 819.642,A -85,B 0,C 180,E1 19057.498,E2 19057.498} C_VEL
LIN {X 0,Y 421.944,Z 774.85,A -85,B 0,C 180,E1 19053.162,E2 19053.162} C_VEL
LIN {X 0,Y 427.59,Z 740.632,A -85,B 0,C 180,E1 19049.814,E2 19049.814} C_VEL
LIN {X 0,Y 426.052,Z 731.94,A -85,B 0,C 180,E1 19048.045,E2 19048.045} C_VEL
LIN {X 0,Y 424.084,Z 723.467,A -85,B 0,C 180,E1 19045.846,E2 19045.846} C_VEL
LIN {X 0,Y 422.135,Z 716.806,A -85,B 0,C 180,E1 19043.518,E2 19043.518} C_VEL
LIN {X 0,Y 421.076,Z 713.299,A -85,B 0,C 180,E1 19041.808,E2 19041.808} C_VEL
LIN {X 0,Y 420.309,Z 709.803,A -85,B 0,C 180,E1 19039.497,E2 19039.497} C_VEL
LIN {X 0,Y 419.698,Z 710.716,A -85,B 0,C 180,E1 19039.065,E2 19039.065} C_VEL
LIN {X 0,Y 418.582,Z 712.821,A -85,B 0,C 180,E1 19038.386,E2 19038.386} C_VEL
LIN {X 0,Y 413.722,Z 726.083,A -85,B 0,C 180,E1 19035.821,E2 19035.821} C_VEL
LIN {X 0,Y 426.297,Z 752.278,A -85,B 0,C 180,E1 19033.843,E2 19033.843} C_VEL
LIN {X 0,Y 410.732,Z 978.43,A -85,B 0,C 180,E1 19028.642,E2 19028.642} C_VEL
LIN {X 0,Y 408.225,Z 1002.849,A -85,B 0,C 180,E1 19027.822,E2 19027.822} C_VEL
LIN {X 0,Y 405.232,Z 1026.477,A -85,B 0,C 180,E1 19026.749,E2 19026.749} C_VEL
LIN {X 0,Y 402.075,Z 1048.156,A -85,B 0,C 180,E1 19025.495,E2 19025.495} C_VEL
LIN {X 0,Y 398.664,Z 1069.167,A -85,B 0,C 180,E1 19024.005,E2 19024.005} C_VEL
LIN {X 0,Y 395.129,Z 1089.441,A -85,B 0,C 180,E1 19022.269,E2 19022.269} C_VEL
LIN {X 0,Y 391.7,Z 1108.219,A -85,B 0,C 180,E1 19020.357,E2 19020.357} C_VEL
LIN {X 0,Y 388.225,Z 1126.655,A -85,B 0,C 180,E1 19018.117,E2 19018.117} C_VEL
LIN {X 0,Y 385.248,Z 1142.426,A -85,B 0,C 180,E1 19015.848,E2 19015.848} C_VEL
LIN {X 0,Y 382.469,Z 1157.81,A -85,B 0,C 180,E1 19013.248,E2 19013.248} C_VEL
LIN {X 0,Y 380.236,Z 1171.18,A -85,B 0,C 180,E1 19010.578,E2 19010.578} C_VEL
LIN {X 0,Y 378.538,Z 1182.698,A -85,B 0,C 180,E1 19007.84,E2 19007.84} C_VEL
LIN {X 0,Y 377.344,Z 1192.459,A -85,B 0,C 180,E1 19005.049,E2 19005.049} C_VEL
LIN {X 0,Y 376.592,Z 1200.945,A -85,B 0,C 180,E1 19002.106,E2 19002.106} C_VEL
LIN {X 0,Y 376.256,Z 1207.604,A -85,B 0,C 180,E1 18999.173,E2 18999.173} C_VEL
LIN {X 0,Y 376.192,Z 1212.593,A -85,B 0,C 180,E1 18996.227,E2 18996.227} C_VEL
LIN {X 0,Y 376.226,Z 1216.003,A -85,B 0,C 180,E1 18993.35,E2 18993.35} C_VEL
LIN {X 0,Y 376.243,Z 1217.785,A -85,B 0,C 180,E1 18990.455,E2 18990.455} C_VEL
LIN {X 0,Y 376.162,Z 1218.193,A -85,B 0,C 180,E1 18987.56,E2 18987.56} C_VEL
LIN {X 0,Y 376.057,Z 1216.998,A -85,B 0,C 180,E1 18984.658,E2 18984.658} C_VEL
LIN {X 0,Y 376.103,Z 1214.184,A -85,B 0,C 180,E1 18981.5,E2 18981.5} C_VEL
LIN {X 0,Y 376.498,Z 1209.7,A -85,B 0,C 180,E1 18978.354,E2 18978.354} C_VEL
LIN {X 0,Y 377.5,Z 1203.331,A -85,B 0,C 180,E1 18975.11,E2 18975.11} C_VEL
LIN {X 0,Y 379.272,Z 1195.182,A -85,B 0,C 180,E1 18971.873,E2 18971.873} C_VEL
LIN {X 0,Y 381.934,Z 1185.088,A -85,B 0,C 180,E1 18968.658,E2 18968.658} C_VEL
LIN {X 0,Y 385.484,Z 1173.255,A -85,B 0,C 180,E1 18965.572,E2 18965.572} C_VEL
LIN {X 0,Y 390.225,Z 1158.902,A -85,B 0,C 180,E1 18962.45,E2 18962.45} C_VEL
LIN {X 0,Y 395.967,Z 1142.6,A -85,B 0,C 180,E1 18959.497,E2 18959.497} C_VEL
LIN {X 0,Y 402.346,Z 1125.242,A -85,B 0,C 180,E1 18956.855,E2 18956.855} C_VEL
LIN {X 0,Y 409.669,Z 1105.868,A -85,B 0,C 180,E1 18954.37,E2 18954.37} C_VEL
LIN {X 0,Y 417.969,Z 1084.246,A -85,B 0,C 180,E1 18952.06,E2 18952.06} C_VEL
LIN {X 0,Y 426.493,Z 1062.315,A -85,B 0,C 180,E1 18950.117,E2 18950.117} C_VEL
LIN {X 0,Y 435.779,Z 1038.247,A -85,B 0,C 180,E1 18948.373,E2 18948.373} C_VEL
LIN {X 0,Y 444.544,Z 1015.001,A -85,B 0,C 180,E1 18947.036,E2 18947.036} C_VEL
LIN {X 0,Y 453.087,Z 991.055,A -85,B 0,C 180,E1 18945.959,E2 18945.959} C_VEL
LIN {X 0,Y 461.792,Z 963.977,A -85,B 0,C 180,E1 18945.011,E2 18945.011} C_VEL
LIN {X 0,Y 465.398,Z 951.379,A -85,B 0,C 180,E1 18944.615,E2 18944.615} C_VEL
LIN {X 0,Y 458.978,Z 972.629,A -85,B 0,C 180,E1 18943.852,E2 18943.852} C_VEL
LIN {X 0,Y 451.509,Z 994.4,A -85,B 0,C 180,E1 18942.836,E2 18942.836} C_VEL
LIN {X 0,Y 443.313,Z 1016.383,A -85,B 0,C 180,E1 18941.541,E2 18941.541} C_VEL
LIN {X 0,Y 434.413,Z 1039.077,A -85,B 0,C 180,E1 18939.871,E2 18939.871} C_VEL
LIN {X 0,Y 425.858,Z 1060.195,A -85,B 0,C 180,E1 18937.966,E2 18937.966} C_VEL
LIN {X 0,Y 417.527,Z 1080.426,A -85,B 0,C 180,E1 18935.758,E2 18935.758} C_VEL
LIN {X 0,Y 409.731,Z 1099.069,A -85,B 0,C 180,E1 18933.307,E2 18933.307} C_VEL
LIN {X 0,Y 402.555,Z 1116.078,A -85,B 0,C 180,E1 18930.613,E2 18930.613} C_VEL
LIN {X 0,Y 396.104,Z 1131.395,A -85,B 0,C 180,E1 18927.679,E2 18927.679} C_VEL
LIN {X 0,Y 390.785,Z 1144.083,A -85,B 0,C 180,E1 18924.722,E2 18924.722} C_VEL
LIN {X 0,Y 386.454,Z 1154.679,A -85,B 0,C 180,E1 18921.718,E2 18921.718} C_VEL
LIN {X 0,Y 382.941,Z 1163.669,A -85,B 0,C 180,E1 18918.578,E2 18918.578} C_VEL
LIN {X 0,Y 380.323,Z 1170.887,A -85,B 0,C 180,E1 18915.402,E2 18915.402} C_VEL
LIN {X 0,Y 378.408,Z 1176.556,A -85,B 0,C 180,E1 18912.052,E2 18912.052} C_VEL
LIN {X 0,Y 377.248,Z 1180.225,A -85,B 0,C 180,E1 18908.846,E2 18908.846} C_VEL
LIN {X 0,Y 376.579,Z 1182.397,A -85,B 0,C 180,E1 18905.488,E2 18905.488} C_VEL
LIN {X 0,Y 376.284,Z 1182.873,A -85,B 0,C 180,E1 18902.356,E2 18902.356} C_VEL
LIN {X 0,Y 376.186,Z 1181.673,A -85,B 0,C 180,E1 18899.242,E2 18899.242} C_VEL
LIN {X 0,Y 376.181,Z 1178.863,A -85,B 0,C 180,E1 18896.041,E2 18896.041} C_VEL
LIN {X 0,Y 376.347,Z 1174.613,A -85,B 0,C 180,E1 18892.984,E2 18892.984} C_VEL
LIN {X 0,Y 376.762,Z 1168.589,A -85,B 0,C 180,E1 18889.916,E2 18889.916} C_VEL
LIN {X 0,Y 377.565,Z 1160.825,A -85,B 0,C 180,E1 18886.839,E2 18886.839} C_VEL
LIN {X 0,Y 378.778,Z 1151.687,A -85,B 0,C 180,E1 18883.912,E2 18883.912} C_VEL
LIN {X 0,Y 380.523,Z 1140.511,A -85,B 0,C 180,E1 18880.988,E2 18880.988} C_VEL
LIN {X 0,Y 382.721,Z 1127.866,A -85,B 0,C 180,E1 18878.228,E2 18878.228} C_VEL
LIN {X 0,Y 385.489,Z 1112.934,A -85,B 0,C 180,E1 18875.484,E2 18875.484} C_VEL
LIN {X 0,Y 388.521,Z 1097.091,A -85,B 0,C 180,E1 18873.026,E2 18873.026} C_VEL
LIN {X 0,Y 391.743,Z 1080.239,A -85,B 0,C 180,E1 18870.803,E2 18870.803} C_VEL
LIN {X 0,Y 395.26,Z 1061.096,A -85,B 0,C 180,E1 18868.682,E2 18868.682} C_VEL
LIN {X 0,Y 398.665,Z 1041.503,A -85,B 0,C 180,E1 18866.859,E2 18866.859} C_VEL
LIN {X 0,Y 402.087,Z 1020.192,A -85,B 0,C 180,E1 18865.205,E2 18865.205} C_VEL
LIN {X 0,Y 405.301,Z 997.712,A -85,B 0,C 180,E1 18863.779,E2 18863.779} C_VEL
LIN {X 0,Y 408.022,Z 975.924,A -85,B 0,C 180,E1 18862.667,E2 18862.667} C_VEL
LIN {X 0,Y 410.436,Z 952.398,A -85,B 0,C 180,E1 18861.733,E2 18861.733} C_VEL
LIN {X 0,Y 412.336,Z 927.897,A -85,B 0,C 180,E1 18861.036,E2 18861.036} C_VEL
LIN {X 0,Y 425.34,Z 734.497,A -85,B 0,C 180,E1 18856.637,E2 18856.637} C_VEL
LIN {X 0,Y 407.411,Z 702.268,A -85,B 0,C 180,E1 18853.92,E2 18853.92} C_VEL
LIN {X 0,Y 391.039,Z 674.608,A -85,B 0,C 180,E1 18851.231,E2 18851.231} C_VEL
LIN {X 0,Y 380.932,Z 658.018,A -85,B 0,C 180,E1 18849.438,E2 18849.438} C_VEL
LIN {X 0,Y 379.044,Z 654.782,A -85,B 0,C 180,E1 18849.086,E2 18849.086} C_VEL
LIN {X 0,Y 378.776,Z 653.489,A -85,B 0,C 180,E1 18848.965,E2 18848.965} C_VEL
LIN {X 0,Y 378.812,Z 653.475,A -85,B 0,C 180,E1 18844.946,E2 18844.946} C_VEL
LIN {X 0,Y 378.847,Z 653.481,A -85,B 0,C 180,E1 18840.941,E2 18840.941} C_VEL
LIN {X 0,Y 378.835,Z 653.478,A -85,B 0,C 180,E1 18837.001,E2 18837.001} C_VEL
LIN {X 0,Y 378.792,Z 653.48,A -85,B 0,C 180,E1 18832.998,E2 18832.998} C_VEL
LIN {X 0,Y 378.796,Z 653.479,A -85,B 0,C 180,E1 18828.948,E2 18828.948} C_VEL
LIN {X 0,Y 378.828,Z 653.477,A -85,B 0,C 180,E1 18824.993,E2 18824.993} C_VEL
LIN {X 0,Y 378.847,Z 653.478,A -85,B 0,C 180,E1 18820.956,E2 18820.956} C_VEL
LIN {X 0,Y 378.846,Z 653.47,A -85,B 0,C 180,E1 18816.975,E2 18816.975} C_VEL
LIN {X 0,Y 378.798,Z 653.464,A -85,B 0,C 180,E1 18812.877,E2 18812.877} C_VEL
LIN {X 0,Y 378.839,Z 653.477,A -85,B 0,C 180,E1 18808.943,E2 18808.943} C_VEL
LIN {X 0,Y 378.845,Z 653.464,A -85,B 0,C 180,E1 18804.854,E2 18804.854} C_VEL
LIN {X 0,Y 378.836,Z 653.473,A -85,B 0,C 180,E1 18800.89,E2 18800.89} C_VEL
LIN {X 0,Y 378.805,Z 653.47,A -85,B 0,C 180,E1 18796.882,E2 18796.882} C_VEL
LIN {X 0,Y 378.822,Z 653.476,A -85,B 0,C 180,E1 18792.808,E2 18792.808} C_VEL
LIN {X 0,Y 378.853,Z 653.477,A -85,B 0,C 180,E1 18788.805,E2 18788.805} C_VEL
LIN {X 0,Y 378.838,Z 653.476,A -85,B 0,C 180,E1 18784.689,E2 18784.689} C_VEL
LIN {X 0,Y 378.805,Z 653.483,A -85,B 0,C 180,E1 18780.772,E2 18780.772} C_VEL
LIN {X 0,Y 378.786,Z 653.487,A -85,B 0,C 180,E1 18776.7,E2 18776.7} C_VEL
LIN {X 0,Y 378.83,Z 653.481,A -85,B 0,C 180,E1 18772.626,E2 18772.626} C_VEL
LIN {X 0,Y 378.865,Z 653.635,A -85,B 0,C 180,E1 18771.932,E2 18771.932} C_VEL
LIN {X 0,Y 387.503,Z 680.157,A -85,B 0,C 180,E1 18768.562,E2 18768.562} C_VEL
LIN {X 0,Y 394.383,Z 704.082,A -85,B 0,C 180,E1 18765.698,E2 18765.698} C_VEL
LIN {X 0,Y 395.954,Z 710.126,A -85,B 0,C 180,E1 18764.992,E2 18764.992} C_VEL
LIN {X 0,Y 395.104,Z 723.822,A -85,B 0,C 180,E1 18763.709,E2 18763.709} C_VEL
LIN {X 0,Y 393.772,Z 730.435,A -85,B 0,C 180,E1 18763.145,E2 18763.145} C_VEL
LIN {X 0,Y 386.562,Z 749.358,A -85,B 0,C 180,E1 18761.747,E2 18761.747} C_VEL
LIN {X 0,Y 385.749,Z 754.082,A -85,B 0,C 180,E1 18761.332,E2 18761.332} C_VEL
LIN {X 0,Y 382.946,Z 798.914,A -85,B 0,C 180,E1 18757.091,E2 18757.091} C_VEL
LIN {X 0,Y 380.242,Z 845.517,A -85,B 0,C 180,E1 18752.709,E2 18752.709} C_VEL
LIN {X 0,Y 379.881,Z 849.625,A -85,B 0,C 180,E1 18752.383,E2 18752.383} C_VEL
LIN {X 0,Y 375.836,Z 984.958,A -85,B 0,C 180,E1 18748.969,E2 18748.969} C_VEL
LIN {X 0,Y 375.54,Z 1002.913,A -85,B 0,C 180,E1 18748.377,E2 18748.377} C_VEL
LIN {X 0,Y 374.936,Z 1020.889,A -85,B 0,C 180,E1 18747.471,E2 18747.471} C_VEL
LIN {X 0,Y 374.199,Z 1037.162,A -85,B 0,C 180,E1 18746.327,E2 18746.327} C_VEL
LIN {X 0,Y 373.381,Z 1051.568,A -85,B 0,C 180,E1 18745.027,E2 18745.027} C_VEL
LIN {X 0,Y 372.442,Z 1066.315,A -85,B 0,C 180,E1 18743.349,E2 18743.349} C_VEL
LIN {X 0,Y 371.553,Z 1079.381,A -85,B 0,C 180,E1 18741.464,E2 18741.464} C_VEL
LIN {X 0,Y 370.849,Z 1090.171,A -85,B 0,C 180,E1 18739.528,E2 18739.528} C_VEL
LIN {X 0,Y 370.326,Z 1099.49,A -85,B 0,C 180,E1 18737.436,E2 18737.436} C_VEL
LIN {X 0,Y 370.001,Z 1107.265,A -85,B 0,C 180,E1 18735.193,E2 18735.193} C_VEL
LIN {X 0,Y 369.9,Z 1113.468,A -85,B 0,C 180,E1 18732.803,E2 18732.803} C_VEL
LIN {X 0,Y 370.073,Z 1117.845,A -85,B 0,C 180,E1 18730.269,E2 18730.269} C_VEL
LIN {X 0,Y 370.504,Z 1120.136,A -85,B 0,C 180,E1 18727.907,E2 18727.907} C_VEL
LIN {X 0,Y 371.285,Z 1120.619,A -85,B 0,C 180,E1 18725.405,E2 18725.405} C_VEL
LIN {X 0,Y 372.36,Z 1119.361,A -85,B 0,C 180,E1 18723.075,E2 18723.075} C_VEL
LIN {X 0,Y 373.774,Z 1116.296,A -85,B 0,C 180,E1 18720.763,E2 18720.763} C_VEL
LIN {X 0,Y 375.581,Z 1111.474,A -85,B 0,C 180,E1 18718.471,E2 18718.471} C_VEL
LIN {X 0,Y 377.617,Z 1105.126,A -85,B 0,C 180,E1 18716.353,E2 18716.353} C_VEL
LIN {X 0,Y 379.988,Z 1096.776,A -85,B 0,C 180,E1 18714.258,E2 18714.258} C_VEL
LIN {X 0,Y 382.455,Z 1086.868,A -85,B 0,C 180,E1 18712.335,E2 18712.335} C_VEL
LIN {X 0,Y 384.978,Z 1075.503,A -85,B 0,C 180,E1 18710.579,E2 18710.579} C_VEL
LIN {X 0,Y 387.398,Z 1062.386,A -85,B 0,C 180,E1 18708.986,E2 18708.986} C_VEL
LIN {X 0,Y 389.451,Z 1048.986,A -85,B 0,C 180,E1 18707.693,E2 18707.693} C_VEL
LIN {X 0,Y 391.205,Z 1034.874,A -85,B 0,C 180,E1 18706.623,E2 18706.623} C_VEL
LIN {X 0,Y 392.479,Z 1021.799,A -85,B 0,C 180,E1 18705.841,E2 18705.841} C_VEL
LIN {X 0,Y 393.521,Z 1006.917,A -85,B 0,C 180,E1 18705.155,E2 18705.155} C_VEL
LIN {X 0,Y 395.5,Z 969.998,A -85,B 0,C 180,E1 18704.015,E2 18704.015} C_VEL
LIN {X 0,Y 404.107,Z 866.361,A -85,B 0,C 180,E1 18701.084,E2 18701.084} C_VEL
LIN {X 0,Y 410.169,Z 821.178,A -85,B 0,C 180,E1 18696.661,E2 18696.661} C_VEL
LIN {X 0,Y 417.077,Z 777.363,A -85,B 0,C 180,E1 18692.359,E2 18692.359} C_VEL
LIN {X 0,Y 422.832,Z 744.98,A -85,B 0,C 180,E1 18689.123,E2 18689.123} C_VEL
LIN {X 0,Y 421.524,Z 736.778,A -85,B 0,C 180,E1 18687.356,E2 18687.356} C_VEL
LIN {X 0,Y 419.89,Z 729.313,A -85,B 0,C 180,E1 18685.307,E2 18685.307} C_VEL
LIN {X 0,Y 418.477,Z 723.499,A -85,B 0,C 180,E1 18683.147,E2 18683.147} C_VEL
LIN {X 0,Y 417.736,Z 720.512,A -85,B 0,C 180,E1 18681.685,E2 18681.685} C_VEL
LIN {X 0,Y 417.134,Z 717.402,A -85,B 0,C 180,E1 18679.554,E2 18679.554} C_VEL
LIN {X 0,Y 416.16,Z 719.172,A -85,B 0,C 180,E1 18678.972,E2 18678.972} C_VEL
LIN {X 0,Y 410.192,Z 734.696,A -85,B 0,C 180,E1 18675.992,E2 18675.992} C_VEL
LIN {X 0,Y 410.311,Z 735.438,A -85,B 0,C 180,E1 18675.867,E2 18675.867} C_VEL
LIN {X 0,Y 419.462,Z 754.986,A -85,B 0,C 180,E1 18674.389,E2 18674.389} C_VEL
LIN {X 0,Y 403.595,Z 977.979,A -85,B 0,C 180,E1 18669.154,E2 18669.154} C_VEL
LIN {X 0,Y 401.013,Z 1002.483,A -85,B 0,C 180,E1 18668.313,E2 18668.313} C_VEL
LIN {X 0,Y 397.921,Z 1026.214,A -85,B 0,C 180,E1 18667.215,E2 18667.215} C_VEL
LIN {X 0,Y 394.618,Z 1048.302,A -85,B 0,C 180,E1 18665.911,E2 18665.911} C_VEL
LIN {X 0,Y 391.133,Z 1069.198,A -85,B 0,C 180,E1 18664.397,E2 18664.397} C_VEL
LIN {X 0,Y 387.377,Z 1090.164,A -85,B 0,C 180,E1 18662.557,E2 18662.557} C_VEL
LIN {X 0,Y 383.88,Z 1108.77,A -85,B 0,C 180,E1 18660.609,E2 18660.609} C_VEL
LIN {X 0,Y 380.345,Z 1127.136,A -85,B 0,C 180,E1 18658.325,E2 18658.325} C_VEL
LIN {X 0,Y 377.128,Z 1143.78,A -85,B 0,C 180,E1 18655.855,E2 18655.855} C_VEL
LIN {X 0,Y 374.394,Z 1158.606,A -85,B 0,C 180,E1 18653.255,E2 18653.255} C_VEL
LIN {X 0,Y 372.091,Z 1172.152,A -85,B 0,C 180,E1 18650.444,E2 18650.444} C_VEL
LIN {X 0,Y 370.393,Z 1183.697,A -85,B 0,C 180,E1 18647.596,E2 18647.596} C_VEL
LIN {X 0,Y 369.193,Z 1193.724,A -85,B 0,C 180,E1 18644.586,E2 18644.586} C_VEL
LIN {X 0,Y 368.517,Z 1201.823,A -85,B 0,C 180,E1 18641.58,E2 18641.58} C_VEL
LIN {X 0,Y 368.25,Z 1208.225,A -85,B 0,C 180,E1 18638.586,E2 18638.586} C_VEL
LIN {X 0,Y 368.214,Z 1212.873,A -85,B 0,C 180,E1 18635.608,E2 18635.608} C_VEL
LIN {X 0,Y 368.263,Z 1216.077,A -85,B 0,C 180,E1 18632.488,E2 18632.488} C_VEL
LIN {X 0,Y 368.246,Z 1217.525,A -85,B 0,C 180,E1 18629.687,E2 18629.687} C_VEL
LIN {X 0,Y 368.134,Z 1217.522,A -85,B 0,C 180,E1 18626.572,E2 18626.572} C_VEL
LIN {X 0,Y 368.047,Z 1216.073,A -85,B 0,C 180,E1 18623.603,E2 18623.603} C_VEL
LIN {X 0,Y 368.185,Z 1212.786,A -85,B 0,C 180,E1 18620.348,E2 18620.348} C_VEL
LIN {X 0,Y 368.833,Z 1207.729,A -85,B 0,C 180,E1 18616.995,E2 18616.995} C_VEL
LIN {X 0,Y 370.176,Z 1200.945,A -85,B 0,C 180,E1 18613.683,E2 18613.683} C_VEL
LIN {X 0,Y 372.381,Z 1192.284,A -85,B 0,C 180,E1 18610.387,E2 18610.387} C_VEL
LIN {X 0,Y 375.743,Z 1181.201,A -85,B 0,C 180,E1 18606.97,E2 18606.97} C_VEL
LIN {X 0,Y 380.005,Z 1168.74,A -85,B 0,C 180,E1 18603.805,E2 18603.805} C_VEL
LIN {X 0,Y 385.268,Z 1154.502,A -85,B 0,C 180,E1 18600.794,E2 18600.794} C_VEL
LIN {X 0,Y 391.555,Z 1138.216,A -85,B 0,C 180,E1 18597.915,E2 18597.915} C_VEL
LIN {X 0,Y 398.637,Z 1120.596,A -85,B 0,C 180,E1 18595.291,E2 18595.291} C_VEL
LIN {X 0,Y 406.862,Z 1100.719,A -85,B 0,C 180,E1 18592.801,E2 18592.801} C_VEL
LIN {X 0,Y 416.323,Z 1078.275,A -85,B 0,C 180,E1 18590.47,E2 18590.47} C_VEL
LIN {X 0,Y 426.263,Z 1054.944,A -85,B 0,C 180,E1 18588.495,E2 18588.495} C_VEL
LIN {X 0,Y 435.794,Z 1032.409,A -85,B 0,C 180,E1 18586.952,E2 18586.952} C_VEL
LIN {X 0,Y 444.906,Z 1010.237,A -85,B 0,C 180,E1 18585.746,E2 18585.746} C_VEL
LIN {X 0,Y 454.414,Z 985.404,A -85,B 0,C 180,E1 18584.704,E2 18584.704} C_VEL
LIN {X 0,Y 455.863,Z 981.236,A -85,B 0,C 180,E1 18584.537,E2 18584.537} C_VEL
LIN {X 0,Y 447.28,Z 1003.388,A -85,B 0,C 180,E1 18583.428,E2 18583.428} C_VEL
LIN {X 0,Y 437.906,Z 1025.826,A -85,B 0,C 180,E1 18581.994,E2 18581.994} C_VEL
LIN {X 0,Y 428.167,Z 1048.086,A -85,B 0,C 180,E1 18580.213,E2 18580.213} C_VEL
LIN {X 0,Y 418.913,Z 1068.717,A -85,B 0,C 180,E1 18578.187,E2 18578.187} C_VEL
LIN {X 0,Y 410.165,Z 1088.026,A -85,B 0,C 180,E1 18575.897,E2 18575.897} C_VEL
LIN {X 0,Y 402.398,Z 1104.99,A -85,B 0,C 180,E1 18573.482,E2 18573.482} C_VEL
LIN {X 0,Y 395.044,Z 1121.032,A -85,B 0,C 180,E1 18570.752,E2 18570.752} C_VEL
LIN {X 0,Y 388.425,Z 1135.514,A -85,B 0,C 180,E1 18567.774,E2 18567.774} C_VEL
LIN {X 0,Y 382.887,Z 1147.798,A -85,B 0,C 180,E1 18564.701,E2 18564.701} C_VEL
LIN {X 0,Y 378.376,Z 1158.094,A -85,B 0,C 180,E1 18561.553,E2 18561.553} C_VEL
LIN {X 0,Y 374.682,Z 1166.894,A -85,B 0,C 180,E1 18558.185,E2 18558.185} C_VEL
LIN {X 0,Y 371.987,Z 1173.636,A -85,B 0,C 180,E1 18554.798,E2 18554.798} C_VEL
LIN {X 0,Y 370.228,Z 1178.404,A -85,B 0,C 180,E1 18551.532,E2 18551.532} C_VEL
LIN {X 0,Y 369.131,Z 1181.619,A -85,B 0,C 180,E1 18548.257,E2 18548.257} C_VEL
LIN {X 0,Y 368.552,Z 1183.117,A -85,B 0,C 180,E1 18545.14,E2 18545.14} C_VEL
LIN {X 0,Y 368.272,Z 1183.147,A -85,B 0,C 180,E1 18541.87,E2 18541.87} C_VEL
LIN {X 0,Y 368.18,Z 1181.714,A -85,B 0,C 180,E1 18538.758,E2 18538.758} C_VEL
LIN {X 0,Y 368.192,Z 1178.639,A -85,B 0,C 180,E1 18535.643,E2 18535.643} C_VEL
LIN {X 0,Y 368.413,Z 1173.759,A -85,B 0,C 180,E1 18532.361,E2 18532.361} C_VEL
LIN {X 0,Y 368.917,Z 1167.427,A -85,B 0,C 180,E1 18529.225,E2 18529.225} C_VEL
LIN {X 0,Y 369.769,Z 1159.605,A -85,B 0,C 180,E1 18526.238,E2 18526.238} C_VEL
LIN {X 0,Y 371.103,Z 1150.02,A -85,B 0,C 180,E1 18523.248,E2 18523.248} C_VEL
LIN {X 0,Y 372.89,Z 1139.147,A -85,B 0,C 180,E1 18520.42,E2 18520.42} C_VEL
LIN {X 0,Y 375.232,Z 1126.173,A -85,B 0,C 180,E1 18517.605,E2 18517.605} C_VEL
LIN {X 0,Y 377.984,Z 1111.712,A -85,B 0,C 180,E1 18514.964,E2 18514.964} C_VEL
LIN {X 0,Y 381.128,Z 1095.604,A -85,B 0,C 180,E1 18512.469,E2 18512.469} C_VEL
LIN {X 0,Y 384.468,Z 1078.506,A -85,B 0,C 180,E1 18510.22,E2 18510.22} C_VEL
LIN {X 0,Y 388.028,Z 1059.612,A -85,B 0,C 180,E1 18508.117,E2 18508.117} C_VEL
LIN {X 0,Y 391.705,Z 1038.849,A -85,B 0,C 180,E1 18506.192,E2 18506.192} C_VEL
LIN {X 0,Y 395.115,Z 1017.789,A -85,B 0,C 180,E1 18504.576,E2 18504.576} C_VEL
LIN {X 0,Y 398.205,Z 996.43,A -85,B 0,C 180,E1 18503.228,E2 18503.228} C_VEL
LIN {X 0,Y 401.135,Z 972.994,A -85,B 0,C 180,E1 18502.044,E2 18502.044} C_VEL
LIN {X 0,Y 403.489,Z 949.909,A -85,B 0,C 180,E1 18501.144,E2 18501.144} C_VEL
LIN {X 0,Y 405.393,Z 925.897,A -85,B 0,C 180,E1 18500.468,E2 18500.468} C_VEL
LIN {X 0,Y 418.514,Z 737.28,A -85,B 0,C 180,E1 18496.093,E2 18496.093} C_VEL
LIN {X 0,Y 400.598,Z 704.994,A -85,B 0,C 180,E1 18493.298,E2 18493.298} C_VEL
LIN {X 0,Y 383.363,Z 675.863,A -85,B 0,C 180,E1 18490.379,E2 18490.379} C_VEL
LIN {X 0,Y 375.257,Z 662.873,A -85,B 0,C 180,E1 18488.925,E2 18488.925} C_VEL
LIN {X 0,Y 372.691,Z 658.648,A -85,B 0,C 180,E1 18488.447,E2 18488.447} C_VEL
LIN {X 0,Y 371.036,Z 655.318,A -85,B 0,C 180,E1 18488.108,E2 18488.108} C_VEL
LIN {X 0,Y 370.881,Z 654.464,A -85,B 0,C 180,E1 18488.054,E2 18488.054} C_VEL
LIN {X 0,Y 370.903,Z 654.468,A -85,B 0,C 180,E1 18483.877,E2 18483.877} C_VEL
LIN {X 0,Y 370.918,Z 654.459,A -85,B 0,C 180,E1 18479.738,E2 18479.738} C_VEL
LIN {X 0,Y 370.899,Z 654.461,A -85,B 0,C 180,E1 18475.726,E2 18475.726} C_VEL
LIN {X 0,Y 370.878,Z 654.464,A -85,B 0,C 180,E1 18471.558,E2 18471.558} C_VEL
LIN {X 0,Y 370.892,Z 654.46,A -85,B 0,C 180,E1 18467.394,E2 18467.394} C_VEL
LIN {X 0,Y 370.91,Z 654.451,A -85,B 0,C 180,E1 18463.321,E2 18463.321} C_VEL
LIN {X 0,Y 370.908,Z 654.454,A -85,B 0,C 180,E1 18459.154,E2 18459.154} C_VEL
LIN {X 0,Y 370.881,Z 654.472,A -85,B 0,C 180,E1 18455.106,E2 18455.106} C_VEL
LIN {X 0,Y 370.884,Z 654.462,A -85,B 0,C 180,E1 18450.929,E2 18450.929} C_VEL
LIN {X 0,Y 370.901,Z 654.449,A -85,B 0,C 180,E1 18446.911,E2 18446.911} C_VEL
LIN {X 0,Y 370.92,Z 654.463,A -85,B 0,C 180,E1 18442.72,E2 18442.72} C_VEL
LIN {X 0,Y 370.889,Z 654.441,A -85,B 0,C 180,E1 18438.652,E2 18438.652} C_VEL
LIN {X 0,Y 370.88,Z 654.47,A -85,B 0,C 180,E1 18434.522,E2 18434.522} C_VEL
LIN {X 0,Y 370.904,Z 654.464,A -85,B 0,C 180,E1 18430.474,E2 18430.474} C_VEL
LIN {X 0,Y 370.912,Z 654.462,A -85,B 0,C 180,E1 18426.417,E2 18426.417} C_VEL
LIN {X 0,Y 370.897,Z 654.468,A -85,B 0,C 180,E1 18422.377,E2 18422.377} C_VEL
LIN {X 0,Y 370.863,Z 654.474,A -85,B 0,C 180,E1 18418.418,E2 18418.418} C_VEL
LIN {X 0,Y 370.892,Z 654.469,A -85,B 0,C 180,E1 18414.2,E2 18414.2} C_VEL
LIN {X 0,Y 370.91,Z 654.558,A -85,B 0,C 180,E1 18412.495,E2 18412.495} C_VEL
LIN {X 0,Y 379.393,Z 680.395,A -85,B 0,C 180,E1 18409.14,E2 18409.14} C_VEL
LIN {X 0,Y 386.249,Z 703.89,A -85,B 0,C 180,E1 18406.28,E2 18406.28} C_VEL
LIN {X 0,Y 388.439,Z 712.608,A -85,B 0,C 180,E1 18405.266,E2 18405.266} C_VEL
LIN {X 0,Y 385.749,Z 754.082,A -85,B 0,C 180,E1 18401.332,E2 18401.332} C_VEL
LIN {X 0,Y 384.387,Z 760.714,A -85,B 0,C 180,E1 18400.766,E2 18400.766} C_VEL
LIN {X 0,Y 377.358,Z 778.674,A -85,B 0,C 180,E1 18399.416,E2 18399.416} C_VEL
LIN {X 0,Y 376.272,Z 784.371,A -85,B 0,C 180,E1 18398.913,E2 18398.913} C_VEL
LIN {X 0,Y 373.59,Z 827.94,A -85,B 0,C 180,E1 18394.751,E2 18394.751} C_VEL
LIN {X 0,Y 372.126,Z 849.956,A -85,B 0,C 180,E1 18392.681,E2 18392.681} C_VEL
LIN {X 0,Y 367.945,Z 985.246,A -85,B 0,C 180,E1 18389.17,E2 18389.17} C_VEL
LIN {X 0,Y 367.633,Z 1003.53,A -85,B 0,C 180,E1 18388.555,E2 18388.555} C_VEL
LIN {X 0,Y 367.016,Z 1021.355,A -85,B 0,C 180,E1 18387.637,E2 18387.637} C_VEL
LIN {X 0,Y 366.276,Z 1037.411,A -85,B 0,C 180,E1 18386.496,E2 18386.496} C_VEL
LIN {X 0,Y 365.445,Z 1051.92,A -85,B 0,C 180,E1 18385.176,E2 18385.176} C_VEL
LIN {X 0,Y 364.47,Z 1066.992,A -85,B 0,C 180,E1 18383.436,E2 18383.436} C_VEL
LIN {X 0,Y 363.572,Z 1080.057,A -85,B 0,C 180,E1 18381.524,E2 18381.524} C_VEL
LIN {X 0,Y 362.861,Z 1090.915,A -85,B 0,C 180,E1 18379.55,E2 18379.55} C_VEL
LIN {X 0,Y 362.31,Z 1100.801,A -85,B 0,C 180,E1 18377.288,E2 18377.288} C_VEL
LIN {X 0,Y 362.006,Z 1108.378,A -85,B 0,C 180,E1 18375.045,E2 18375.045} C_VEL
LIN {X 0,Y 361.928,Z 1114.552,A -85,B 0,C 180,E1 18372.603,E2 18372.603} C_VEL
LIN {X 0,Y 362.14,Z 1118.912,A -85,B 0,C 180,E1 18370.014,E2 18370.014} C_VEL
LIN {X 0,Y 362.629,Z 1121.213,A -85,B 0,C 180,E1 18367.602,E2 18367.602} C_VEL
LIN {X 0,Y 363.496,Z 1121.698,A -85,B 0,C 180,E1 18365.046,E2 18365.046} C_VEL
LIN {X 0,Y 364.668,Z 1120.437,A -85,B 0,C 180,E1 18362.668,E2 18362.668} C_VEL
LIN {X 0,Y 366.211,Z 1117.399,A -85,B 0,C 180,E1 18360.309,E2 18360.309} C_VEL
LIN {X 0,Y 368.172,Z 1112.543,A -85,B 0,C 180,E1 18357.962,E2 18357.962} C_VEL
LIN {X 0,Y 370.342,Z 1106.189,A -85,B 0,C 180,E1 18355.816,E2 18355.816} C_VEL
LIN {X 0,Y 372.892,Z 1097.895,A -85,B 0,C 180,E1 18353.685,E2 18353.685} C_VEL
LIN {X 0,Y 375.526,Z 1088.019,A -85,B 0,C 180,E1 18351.73,E2 18351.73} C_VEL
LIN {X 0,Y 378.195,Z 1076.609,A -85,B 0,C 180,E1 18349.948,E2 18349.948} C_VEL
LIN {X 0,Y 381.022,Z 1062.258,A -85,B 0,C 180,E1 18348.186,E2 18348.186} C_VEL
LIN {X 0,Y 383.352,Z 1047.78,A -85,B 0,C 180,E1 18346.804,E2 18346.804} C_VEL
LIN {X 0,Y 385.082,Z 1034.064,A -85,B 0,C 180,E1 18345.793,E2 18345.793} C_VEL
LIN {X 0,Y 386.359,Z 1021.161,A -85,B 0,C 180,E1 18345.037,E2 18345.037} C_VEL
LIN {X 0,Y 387.545,Z 1004.219,A -85,B 0,C 180,E1 18344.284,E2 18344.284} C_VEL
LIN {X 0,Y 390.144,Z 963.706,A -85,B 0,C 180,E1 18343.033,E2 18343.033} C_VEL
LIN {X 0,Y 398.645,Z 868.259,A -85,B 0,C 180,E1 18340.281,E2 18340.281} C_VEL
LIN {X 0,Y 405.197,Z 822.293,A -85,B 0,C 180,E1 18335.738,E2 18335.738} C_VEL
LIN {X 0,Y 412.903,Z 777.381,A -85,B 0,C 180,E1 18331.267,E2 18331.267} C_VEL
LIN {X 0,Y 418.21,Z 749.84,A -85,B 0,C 180,E1 18328.503,E2 18328.503} C_VEL
LIN {X 0,Y 417.171,Z 741.946,A -85,B 0,C 180,E1 18326.707,E2 18326.707} C_VEL
LIN {X 0,Y 415.92,Z 735.294,A -85,B 0,C 180,E1 18324.759,E2 18324.759} C_VEL
LIN {X 0,Y 414.791,Z 730.036,A -85,B 0,C 180,E1 18322.698,E2 18322.698} C_VEL
LIN {X 0,Y 414.273,Z 727.406,A -85,B 0,C 180,E1 18321.306,E2 18321.306} C_VEL
LIN {X 0,Y 413.949,Z 725.129,A -85,B 0,C 180,E1 18319.692,E2 18319.692} C_VEL
LIN {X 0,Y 409.445,Z 735.039,A -85,B 0,C 180,E1 18317.723,E2 18317.723} C_VEL
LIN {X 0,Y 406.546,Z 744.203,A -85,B 0,C 180,E1 18315.961,E2 18315.961} C_VEL
LIN {X 0,Y 412.663,Z 757.581,A -85,B 0,C 180,E1 18314.954,E2 18314.954} C_VEL
LIN {X 0,Y 396.414,Z 977.886,A -85,B 0,C 180,E1 18309.659,E2 18309.659} C_VEL
LIN {X 0,Y 393.753,Z 1002.471,A -85,B 0,C 180,E1 18308.798,E2 18308.798} C_VEL
LIN {X 0,Y 390.547,Z 1026.437,A -85,B 0,C 180,E1 18307.665,E2 18307.665} C_VEL
LIN {X 0,Y 387.164,Z 1048.431,A -85,B 0,C 180,E1 18306.337,E2 18306.337} C_VEL
LIN {X 0,Y 383.619,Z 1069.137,A -85,B 0,C 180,E1 18304.804,E2 18304.804} C_VEL
LIN {X 0,Y 379.776,Z 1090.052,A -85,B 0,C 180,E1 18302.932,E2 18302.932} C_VEL
LIN {X 0,Y 376.199,Z 1108.624,A -85,B 0,C 180,E1 18300.948,E2 18300.948} C_VEL
LIN {X 0,Y 372.637,Z 1126.673,A -85,B 0,C 180,E1 18298.661,E2 18298.661} C_VEL
LIN {X 0,Y 369.381,Z 1143.112,A -85,B 0,C 180,E1 18296.18,E2 18296.18} C_VEL
LIN {X 0,Y 366.633,Z 1157.636,A -85,B 0,C 180,E1 18293.597,E2 18293.597} C_VEL
LIN {X 0,Y 364.255,Z 1171.255,A -85,B 0,C 180,E1 18290.736,E2 18290.736} C_VEL
LIN {X 0,Y 362.489,Z 1182.898,A -85,B 0,C 180,E1 18287.827,E2 18287.827} C_VEL
LIN {X 0,Y 361.243,Z 1192.98,A -85,B 0,C 180,E1 18284.75,E2 18284.75} C_VEL
LIN {X 0,Y 360.542,Z 1201.161,A -85,B 0,C 180,E1 18281.678,E2 18281.678} C_VEL
LIN {X 0,Y 360.268,Z 1207.632,A -85,B 0,C 180,E1 18278.617,E2 18278.617} C_VEL
LIN {X 0,Y 360.237,Z 1212.308,A -85,B 0,C 180,E1 18275.573,E2 18275.573} C_VEL
LIN {X 0,Y 360.281,Z 1215.457,A -85,B 0,C 180,E1 18272.543,E2 18272.543} C_VEL
LIN {X 0,Y 360.273,Z 1216.919,A -85,B 0,C 180,E1 18269.839,E2 18269.839} C_VEL
LIN {X 0,Y 360.15,Z 1217.209,A -85,B 0,C 180,E1 18266.815,E2 18266.815} C_VEL
LIN {X 0,Y 360.055,Z 1215.931,A -85,B 0,C 180,E1 18263.78,E2 18263.78} C_VEL
LIN {X 0,Y 360.178,Z 1212.939,A -85,B 0,C 180,E1 18260.41,E2 18260.41} C_VEL
LIN {X 0,Y 360.776,Z 1208.49,A -85,B 0,C 180,E1 18257.188,E2 18257.188} C_VEL
LIN {X 0,Y 362.11,Z 1202.093,A -85,B 0,C 180,E1 18253.804,E2 18253.804} C_VEL
LIN {X 0,Y 364.345,Z 1193.967,A -85,B 0,C 180,E1 18250.437,E2 18250.437} C_VEL
LIN {X 0,Y 367.58,Z 1183.962,A -85,B 0,C 180,E1 18247.107,E2 18247.107} C_VEL
LIN {X 0,Y 371.929,Z 1171.981,A -85,B 0,C 180,E1 18243.837,E2 18243.837} C_VEL
LIN {X 0,Y 377.772,Z 1157.234,A -85,B 0,C 180,E1 18240.506,E2 18240.506} C_VEL
LIN {X 0,Y 384.618,Z 1140.885,A -85,B 0,C 180,E1 18237.441,E2 18237.441} C_VEL
LIN {X 0,Y 392.4,Z 1123.125,A -85,B 0,C 180,E1 18234.658,E2 18234.658} C_VEL
LIN {X 0,Y 401.214,Z 1103.581,A -85,B 0,C 180,E1 18232.096,E2 18232.096} C_VEL
LIN {X 0,Y 411.074,Z 1082.231,A -85,B 0,C 180,E1 18229.773,E2 18229.773} C_VEL
LIN {X 0,Y 421.679,Z 1059.584,A -85,B 0,C 180,E1 18227.758,E2 18227.758} C_VEL
LIN {X 0,Y 432.204,Z 1036.937,A -85,B 0,C 180,E1 18226.14,E2 18226.14} C_VEL
LIN {X 0,Y 441.971,Z 1015.255,A -85,B 0,C 180,E1 18224.917,E2 18224.917} C_VEL
LIN {X 0,Y 446.34,Z 1005.184,A -85,B 0,C 180,E1 18224.429,E2 18224.429} C_VEL
LIN {X 0,Y 436.112,Z 1027.505,A -85,B 0,C 180,E1 18223.01,E2 18223.01} C_VEL
LIN {X 0,Y 425.563,Z 1049.437,A -85,B 0,C 180,E1 18221.246,E2 18221.246} C_VEL
LIN {X 0,Y 415.643,Z 1069.577,A -85,B 0,C 180,E1 18219.251,E2 18219.251} C_VEL
LIN {X 0,Y 406.054,Z 1088.86,A -85,B 0,C 180,E1 18216.933,E2 18216.933} C_VEL
LIN {X 0,Y 397.557,Z 1105.906,A -85,B 0,C 180,E1 18214.467,E2 18214.467} C_VEL
LIN {X 0,Y 389.691,Z 1121.637,A -85,B 0,C 180,E1 18211.739,E2 18211.739} C_VEL
LIN {X 0,Y 382.582,Z 1135.924,A -85,B 0,C 180,E1 18208.747,E2 18208.747} C_VEL
LIN {X 0,Y 376.855,Z 1147.601,A -85,B 0,C 180,E1 18205.797,E2 18205.797} C_VEL
LIN {X 0,Y 371.683,Z 1158.38,A -85,B 0,C 180,E1 18202.461,E2 18202.461} C_VEL
LIN {X 0,Y 367.619,Z 1167.103,A -85,B 0,C 180,E1 18199.053,E2 18199.053} C_VEL
LIN {X 0,Y 364.723,Z 1173.629,A -85,B 0,C 180,E1 18195.751,E2 18195.751} C_VEL
LIN {X 0,Y 362.539,Z 1178.916,A -85,B 0,C 180,E1 18192.103,E2 18192.103} C_VEL
LIN {X 0,Y 361.303,Z 1182.114,A -85,B 0,C 180,E1 18188.758,E2 18188.758} C_VEL
LIN {X 0,Y 360.611,Z 1183.645,A -85,B 0,C 180,E1 18185.413,E2 18185.413} C_VEL
LIN {X 0,Y 360.288,Z 1183.589,A -85,B 0,C 180,E1 18182.071,E2 18182.071} C_VEL
LIN {X 0,Y 360.19,Z 1182.091,A -85,B 0,C 180,E1 18178.89,E2 18178.89} C_VEL
LIN {X 0,Y 360.19,Z 1179.138,A -85,B 0,C 180,E1 18175.865,E2 18175.865} C_VEL
LIN {X 0,Y 360.382,Z 1174.561,A -85,B 0,C 180,E1 18172.671,E2 18172.671} C_VEL
LIN {X 0,Y 360.862,Z 1168.297,A -85,B 0,C 180,E1 18169.466,E2 18169.466} C_VEL
LIN {X 0,Y 361.697,Z 1160.578,A -85,B 0,C 180,E1 18166.414,E2 18166.414} C_VEL
LIN {X 0,Y 363.108,Z 1150.555,A -85,B 0,C 180,E1 18163.198,E2 18163.198} C_VEL
LIN {X 0,Y 364.929,Z 1139.696,A -85,B 0,C 180,E1 18160.309,E2 18160.309} C_VEL
LIN {X 0,Y 367.32,Z 1126.713,A -85,B 0,C 180,E1 18157.434,E2 18157.434} C_VEL
LIN {X 0,Y 370.134,Z 1112.254,A -85,B 0,C 180,E1 18154.738,E2 18154.738} C_VEL
LIN {X 0,Y 373.415,Z 1095.842,A -85,B 0,C 180,E1 18152.148,E2 18152.148} C_VEL
LIN {X 0,Y 376.894,Z 1078.429,A -85,B 0,C 180,E1 18149.823,E2 18149.823} C_VEL
LIN {X 0,Y 380.418,Z 1060.192,A -85,B 0,C 180,E1 18147.758,E2 18147.758} C_VEL
LIN {X 0,Y 384.179,Z 1039.449,A -85,B 0,C 180,E1 18145.798,E2 18145.798} C_VEL
LIN {X 0,Y 387.646,Z 1018.591,A -85,B 0,C 180,E1 18144.165,E2 18144.165} C_VEL
LIN {X 0,Y 390.919,Z 996.55,A -85,B 0,C 180,E1 18142.748,E2 18142.748} C_VEL
LIN {X 0,Y 393.91,Z 973.187,A -85,B 0,C 180,E1 18141.55,E2 18141.55} C_VEL
LIN {X 0,Y 396.328,Z 950.038,A -85,B 0,C 180,E1 18140.633,E2 18140.633} C_VEL
LIN {X 0,Y 398.302,Z 925.822,A -85,B 0,C 180,E1 18139.939,E2 18139.939} C_VEL
LIN {X 0,Y 411.76,Z 740.116,A -85,B 0,C 180,E1 18135.532,E2 18135.532} C_VEL
LIN {X 0,Y 394.488,Z 709.055,A -85,B 0,C 180,E1 18132.79,E2 18132.79} C_VEL
LIN {X 0,Y 378.07,Z 681.125,A -85,B 0,C 180,E1 18129.943,E2 18129.943} C_VEL
LIN {X 0,Y 365.694,Z 660.676,A -85,B 0,C 180,E1 18127.622,E2 18127.622} C_VEL
LIN {X 0,Y 363.39,Z 657.357,A -85,B 0,C 180,E1 18127.181,E2 18127.181} C_VEL
LIN {X 0,Y 362.914,Z 655.46,A -85,B 0,C 180,E1 18127.006,E2 18127.006} C_VEL
LIN {X 0,Y 362.957,Z 655.451,A -85,B 0,C 180,E1 18122.844,E2 18122.844} C_VEL
LIN {X 0,Y 362.969,Z 655.451,A -85,B 0,C 180,E1 18118.823,E2 18118.823} C_VEL
LIN {X 0,Y 362.925,Z 655.466,A -85,B 0,C 180,E1 18114.619,E2 18114.619} C_VEL
LIN {X 0,Y 362.903,Z 655.466,A -85,B 0,C 180,E1 18110.316,E2 18110.316} C_VEL
LIN {X 0,Y 362.955,Z 655.457,A -85,B 0,C 180,E1 18106.157,E2 18106.157} C_VEL
LIN {X 0,Y 362.964,Z 655.451,A -85,B 0,C 180,E1 18102.076,E2 18102.076} C_VEL
LIN {X 0,Y 362.935,Z 655.445,A -85,B 0,C 180,E1 18097.92,E2 18097.92} C_VEL
LIN {X 0,Y 362.898,Z 655.454,A -85,B 0,C 180,E1 18093.794,E2 18093.794} C_VEL
LIN {X 0,Y 362.937,Z 655.46,A -85,B 0,C 180,E1 18089.651,E2 18089.651} C_VEL
LIN {X 0,Y 362.962,Z 655.433,A -85,B 0,C 180,E1 18085.578,E2 18085.578} C_VEL
LIN {X 0,Y 362.947,Z 655.453,A -85,B 0,C 180,E1 18081.447,E2 18081.447} C_VEL
LIN {X 0,Y 362.909,Z 655.447,A -85,B 0,C 180,E1 18077.269,E2 18077.269} C_VEL
LIN {X 0,Y 362.919,Z 655.457,A -85,B 0,C 180,E1 18073.187,E2 18073.187} C_VEL
LIN {X 0,Y 362.962,Z 655.453,A -85,B 0,C 180,E1 18069.187,E2 18069.187} C_VEL
LIN {X 0,Y 362.96,Z 655.456,A -85,B 0,C 180,E1 18065.074,E2 18065.074} C_VEL
LIN {X 0,Y 362.927,Z 655.461,A -85,B 0,C 180,E1 18060.998,E2 18060.998} C_VEL
LIN {X 0,Y 362.906,Z 655.465,A -85,B 0,C 180,E1 18056.753,E2 18056.753} C_VEL
LIN {X 0,Y 362.945,Z 655.533,A -85,B 0,C 180,E1 18053.067,E2 18053.067} C_VEL
LIN {X 0,Y 371.511,Z 681.307,A -85,B 0,C 180,E1 18049.666,E2 18049.666} C_VEL
LIN {X 0,Y 378.446,Z 704.942,A -85,B 0,C 180,E1 18046.719,E2 18046.719} C_VEL
LIN {X 0,Y 380.894,Z 714.768,A -85,B 0,C 180,E1 18045.558,E2 18045.558} C_VEL
LIN {X 0,Y 378.057,Z 757.389,A -85,B 0,C 180,E1 18041.488,E2 18041.488} C_VEL
LIN {X 0,Y 376.272,Z 784.371,A -85,B 0,C 180,E1 18038.913,E2 18038.913} C_VEL
LIN {X 0,Y 374.896,Z 791.021,A -85,B 0,C 180,E1 18038.334,E2 18038.334} C_VEL
LIN {X 0,Y 367.814,Z 808.932,A -85,B 0,C 180,E1 18036.942,E2 18036.942} C_VEL
LIN {X 0,Y 366.739,Z 814.633,A -85,B 0,C 180,E1 18036.428,E2 18036.428} C_VEL
LIN {X 0,Y 364.531,Z 849.578,A -85,B 0,C 180,E1 18033.078,E2 18033.078} C_VEL
LIN {X 0,Y 364.315,Z 851.99,A -85,B 0,C 180,E1 18032.947,E2 18032.947} C_VEL
LIN {X 0,Y 360.052,Z 985.326,A -85,B 0,C 180,E1 18029.374,E2 18029.374} C_VEL
LIN {X 0,Y 359.722,Z 1004.211,A -85,B 0,C 180,E1 18028.732,E2 18028.732} C_VEL
LIN {X 0,Y 359.089,Z 1022.037,A -85,B 0,C 180,E1 18027.797,E2 18027.797} C_VEL
LIN {X 0,Y 358.314,Z 1038.493,A -85,B 0,C 180,E1 18026.603,E2 18026.603} C_VEL
LIN {X 0,Y 357.459,Z 1053.055,A -85,B 0,C 180,E1 18025.246,E2 18025.246} C_VEL
LIN {X 0,Y 356.477,Z 1067.979,A -85,B 0,C 180,E1 18023.486,E2 18023.486} C_VEL
LIN {X 0,Y 355.566,Z 1081.111,A -85,B 0,C 180,E1 18021.525,E2 18021.525} C_VEL
LIN {X 0,Y 354.875,Z 1091.585,A -85,B 0,C 180,E1 18019.586,E2 18019.586} C_VEL
LIN {X 0,Y 354.308,Z 1101.669,A -85,B 0,C 180,E1 18017.233,E2 18017.233} C_VEL
LIN {X 0,Y 354.008,Z 1109.413,A -85,B 0,C 180,E1 18014.89,E2 18014.89} C_VEL
LIN {X 0,Y 353.955,Z 1115.608,A -85,B 0,C 180,E1 18012.394,E2 18012.394} C_VEL
LIN {X 0,Y 354.213,Z 1119.987,A -85,B 0,C 180,E1 18009.747,E2 18009.747} C_VEL
LIN {X 0,Y 354.775,Z 1122.304,A -85,B 0,C 180,E1 18007.246,E2 18007.246} C_VEL
LIN {X 0,Y 355.721,Z 1122.787,A -85,B 0,C 180,E1 18004.672,E2 18004.672} C_VEL
LIN {X 0,Y 357.001,Z 1121.549,A -85,B 0,C 180,E1 18002.244,E2 18002.244} C_VEL
LIN {X 0,Y 358.675,Z 1118.509,A -85,B 0,C 180,E1 17999.837,E2 17999.837} C_VEL
LIN {X 0,Y 360.778,Z 1113.687,A -85,B 0,C 180,E1 17997.455,E2 17997.455} C_VEL
LIN {X 0,Y 363.228,Z 1107.083,A -85,B 0,C 180,E1 17995.174,E2 17995.174} C_VEL
LIN {X 0,Y 365.85,Z 1099.072,A -85,B 0,C 180,E1 17993.09,E2 17993.09} C_VEL
LIN {X 0,Y 368.642,Z 1089.171,A -85,B 0,C 180,E1 17991.103,E2 17991.103} C_VEL
LIN {X 0,Y 371.505,Z 1077.894,A -85,B 0,C 180,E1 17989.294,E2 17989.294} C_VEL
LIN {X 0,Y 374.373,Z 1064.257,A -85,B 0,C 180,E1 17987.581,E2 17987.581} C_VEL
LIN {X 0,Y 376.702,Z 1050.833,A -85,B 0,C 180,E1 17986.254,E2 17986.254} C_VEL
LIN {X 0,Y 378.687,Z 1036.718,A -85,B 0,C 180,E1 17985.157,E2 17985.157} C_VEL
LIN {X 0,Y 380.139,Z 1023.742,A -85,B 0,C 180,E1 17984.356,E2 17984.356} C_VEL
LIN {X 0,Y 381.34,Z 1008.945,A -85,B 0,C 180,E1 17983.651,E2 17983.651} C_VEL
LIN {X 0,Y 383.737,Z 971.696,A -85,B 0,C 180,E1 17982.438,E2 17982.438} C_VEL
LIN {X 0,Y 393.297,Z 869.986,A -85,B 0,C 180,E1 17979.439,E2 17979.439} C_VEL
LIN {X 0,Y 400.162,Z 824.99,A -85,B 0,C 180,E1 17974.939,E2 17974.939} C_VEL
LIN {X 0,Y 408.546,Z 779.643,A -85,B 0,C 180,E1 17970.368,E2 17970.368} C_VEL
LIN {X 0,Y 413.795,Z 754.508,A -85,B 0,C 180,E1 17967.793,E2 17967.793} C_VEL
LIN {X 0,Y 412.963,Z 747.021,A -85,B 0,C 180,E1 17965.989,E2 17965.989} C_VEL
LIN {X 0,Y 411.955,Z 740.478,A -85,B 0,C 180,E1 17963.921,E2 17963.921} C_VEL
LIN {X 0,Y 411.207,Z 736.2,A -85,B 0,C 180,E1 17962.031,E2 17962.031} C_VEL
LIN {X 0,Y 410.889,Z 734.31,A -85,B 0,C 180,E1 17960.917,E2 17960.917} C_VEL
LIN {X 0,Y 410.787,Z 732.983,A -85,B 0,C 180,E1 17959.949,E2 17959.949} C_VEL
LIN {X 0,Y 404.58,Z 747.316,A -85,B 0,C 180,E1 17957.181,E2 17957.181} C_VEL
LIN {X 0,Y 402.926,Z 753.356,A -85,B 0,C 180,E1 17956.032,E2 17956.032} C_VEL
LIN {X 0,Y 405.862,Z 760.011,A -85,B 0,C 180,E1 17955.531,E2 17955.531} C_VEL
LIN {X 0,Y 389.309,Z 977.193,A -85,B 0,C 180,E1 17950.198,E2 17950.198} C_VEL
LIN {X 0,Y 386.582,Z 1001.804,A -85,B 0,C 180,E1 17949.319,E2 17949.319} C_VEL
LIN {X 0,Y 383.408,Z 1024.917,A -85,B 0,C 180,E1 17948.214,E2 17948.214} C_VEL
LIN {X 0,Y 379.95,Z 1047.062,A -85,B 0,C 180,E1 17946.868,E2 17946.868} C_VEL
LIN {X 0,Y 376.124,Z 1068.923,A -85,B 0,C 180,E1 17945.228,E2 17945.228} C_VEL
LIN {X 0,Y 372.212,Z 1089.693,A -85,B 0,C 180,E1 17943.333,E2 17943.333} C_VEL
LIN {X 0,Y 368.451,Z 1108.737,A -85,B 0,C 180,E1 17941.254,E2 17941.254} C_VEL
LIN {X 0,Y 364.87,Z 1126.454,A -85,B 0,C 180,E1 17938.962,E2 17938.962} C_VEL
LIN {X 0,Y 361.55,Z 1142.836,A -85,B 0,C 180,E1 17936.437,E2 17936.437} C_VEL
LIN {X 0,Y 358.771,Z 1157.184,A -85,B 0,C 180,E1 17933.833,E2 17933.833} C_VEL
LIN {X 0,Y 356.427,Z 1170.283,A -85,B 0,C 180,E1 17931.041,E2 17931.041} C_VEL
LIN {X 0,Y 354.592,Z 1182.011,A -85,B 0,C 180,E1 17928.068,E2 17928.068} C_VEL
LIN {X 0,Y 353.297,Z 1192.197,A -85,B 0,C 180,E1 17924.922,E2 17924.922} C_VEL
LIN {X 0,Y 352.57,Z 1200.476,A -85,B 0,C 180,E1 17921.78,E2 17921.78} C_VEL
LIN {X 0,Y 352.287,Z 1207.009,A -85,B 0,C 180,E1 17918.649,E2 17918.649} C_VEL
LIN {X 0,Y 352.261,Z 1211.724,A -85,B 0,C 180,E1 17915.536,E2 17915.536} C_VEL
LIN {X 0,Y 352.306,Z 1214.935,A -85,B 0,C 180,E1 17912.438,E2 17912.438} C_VEL
LIN {X 0,Y 352.279,Z 1216.47,A -85,B 0,C 180,E1 17909.51,E2 17909.51} C_VEL
LIN {X 0,Y 352.148,Z 1216.713,A -85,B 0,C 180,E1 17906.416,E2 17906.416} C_VEL
LIN {X 0,Y 352.048,Z 1215.403,A -85,B 0,C 180,E1 17903.311,E2 17903.311} C_VEL
LIN {X 0,Y 352.238,Z 1212.383,A -85,B 0,C 180,E1 17899.861,E2 17899.861} C_VEL
LIN {X 0,Y 352.959,Z 1207.924,A -85,B 0,C 180,E1 17896.566,E2 17896.566} C_VEL
LIN {X 0,Y 354.486,Z 1201.542,A -85,B 0,C 180,E1 17893.108,E2 17893.108} C_VEL
LIN {X 0,Y 357.117,Z 1193.016,A -85,B 0,C 180,E1 17889.512,E2 17889.512} C_VEL
LIN {X 0,Y 360.938,Z 1182.519,A -85,B 0,C 180,E1 17885.967,E2 17885.967} C_VEL
LIN {X 0,Y 366.026,Z 1169.866,A -85,B 0,C 180,E1 17882.504,E2 17882.504} C_VEL
LIN {X 0,Y 372.171,Z 1155.753,A -85,B 0,C 180,E1 17879.304,E2 17879.304} C_VEL
LIN {X 0,Y 379.63,Z 1139.563,A -85,B 0,C 180,E1 17876.236,E2 17876.236} C_VEL
LIN {X 0,Y 388.456,Z 1121.133,A -85,B 0,C 180,E1 17873.331,E2 17873.331} C_VEL
LIN {X 0,Y 398.229,Z 1101.406,A -85,B 0,C 180,E1 17870.746,E2 17870.746} C_VEL
LIN {X 0,Y 408.824,Z 1080.55,A -85,B 0,C 180,E1 17868.484,E2 17868.484} C_VEL
LIN {X 0,Y 420.4,Z 1058.068,A -85,B 0,C 180,E1 17866.507,E2 17866.507} C_VEL
LIN {X 0,Y 430.936,Z 1037.361,A -85,B 0,C 180,E1 17865.046,E2 17865.046} C_VEL
LIN {X 0,Y 436.908,Z 1025.343,A -85,B 0,C 180,E1 17864.316,E2 17864.316} C_VEL
LIN {X 0,Y 425.986,Z 1046.222,A -85,B 0,C 180,E1 17862.718,E2 17862.718} C_VEL
LIN {X 0,Y 414.669,Z 1067.194,A -85,B 0,C 180,E1 17860.715,E2 17860.715} C_VEL
LIN {X 0,Y 404.002,Z 1086.785,A -85,B 0,C 180,E1 17858.408,E2 17858.408} C_VEL
LIN {X 0,Y 394.274,Z 1104.611,A -85,B 0,C 180,E1 17855.864,E2 17855.864} C_VEL
LIN {X 0,Y 385.326,Z 1121.02,A -85,B 0,C 180,E1 17853.023,E2 17853.023} C_VEL
LIN {X 0,Y 377.592,Z 1135.294,A -85,B 0,C 180,E1 17850.035,E2 17850.035} C_VEL
LIN {X 0,Y 371.028,Z 1147.549,A -85,B 0,C 180,E1 17846.923,E2 17846.923} C_VEL
LIN {X 0,Y 365.258,Z 1158.47,A -85,B 0,C 180,E1 17843.497,E2 17843.497} C_VEL
LIN {X 0,Y 360.836,Z 1167.044,A -85,B 0,C 180,E1 17840.1,E2 17840.1} C_VEL
LIN {X 0,Y 357.44,Z 1173.959,A -85,B 0,C 180,E1 17836.582,E2 17836.582} C_VEL
LIN {X 0,Y 355.017,Z 1179.17,A -85,B 0,C 180,E1 17832.963,E2 17832.963} C_VEL
LIN {X 0,Y 353.541,Z 1182.529,A -85,B 0,C 180,E1 17829.445,E2 17829.445} C_VEL
LIN {X 0,Y 352.725,Z 1184.089,A -85,B 0,C 180,E1 17826.024,E2 17826.024} C_VEL
LIN {X 0,Y 352.329,Z 1184.118,A -85,B 0,C 180,E1 17822.592,E2 17822.592} C_VEL
LIN {X 0,Y 352.205,Z 1182.771,A -85,B 0,C 180,E1 17819.516,E2 17819.516} C_VEL
LIN {X 0,Y 352.19,Z 1179.813,A -85,B 0,C 180,E1 17816.26,E2 17816.26} C_VEL
LIN {X 0,Y 352.351,Z 1175.342,A -85,B 0,C 180,E1 17812.995,E2 17812.995} C_VEL
LIN {X 0,Y 352.764,Z 1169.468,A -85,B 0,C 180,E1 17809.882,E2 17809.882} C_VEL
LIN {X 0,Y 353.633,Z 1161.463,A -85,B 0,C 180,E1 17806.575,E2 17806.575} C_VEL
LIN {X 0,Y 354.941,Z 1152.182,A -85,B 0,C 180,E1 17803.474,E2 17803.474} C_VEL
LIN {X 0,Y 356.849,Z 1140.844,A -85,B 0,C 180,E1 17800.356,E2 17800.356} C_VEL
LIN {X 0,Y 359.255,Z 1127.943,A -85,B 0,C 180,E1 17797.417,E2 17797.417} C_VEL
LIN {X 0,Y 362.1,Z 1113.63,A -85,B 0,C 180,E1 17794.663,E2 17794.663} C_VEL
LIN {X 0,Y 365.429,Z 1097.383,A -85,B 0,C 180,E1 17792.018,E2 17792.018} C_VEL
LIN {X 0,Y 368.958,Z 1080.168,A -85,B 0,C 180,E1 17789.645,E2 17789.645} C_VEL
LIN {X 0,Y 372.676,Z 1061.354,A -85,B 0,C 180,E1 17787.461,E2 17787.461} C_VEL
LIN {X 0,Y 376.357,Z 1041.595,A -85,B 0,C 180,E1 17785.541,E2 17785.541} C_VEL
LIN {X 0,Y 379.883,Z 1021.129,A -85,B 0,C 180,E1 17783.877,E2 17783.877} C_VEL
LIN {X 0,Y 383.319,Z 998.857,A -85,B 0,C 180,E1 17782.387,E2 17782.387} C_VEL
LIN {X 0,Y 386.257,Z 977.153,A -85,B 0,C 180,E1 17781.216,E2 17781.216} C_VEL
LIN {X 0,Y 388.913,Z 953.396,A -85,B 0,C 180,E1 17780.216,E2 17780.216} C_VEL
LIN {X 0,Y 391.036,Z 928.472,A -85,B 0,C 180,E1 17779.46,E2 17779.46} C_VEL
LIN {X 0,Y 404.893,Z 742.809,A -85,B 0,C 180,E1 17774.96,E2 17774.96} C_VEL
LIN {X 0,Y 387.111,Z 710.737,A -85,B 0,C 180,E1 17772.04,E2 17772.04} C_VEL
LIN {X 0,Y 370.742,Z 683.063,A -85,B 0,C 180,E1 17769.133,E2 17769.133} C_VEL
LIN {X 0,Y 359.539,Z 664.975,A -85,B 0,C 180,E1 17766.972,E2 17766.972} C_VEL
LIN {X 0,Y 357.055,Z 660.883,A -85,B 0,C 180,E1 17766.471,E2 17766.471} C_VEL
LIN {X 0,Y 355.237,Z 657.567,A -85,B 0,C 180,E1 17766.087,E2 17766.087} C_VEL
LIN {X 0,Y 355.012,Z 656.443,A -85,B 0,C 180,E1 17765.969,E2 17765.969} C_VEL
LIN {X 0,Y 355.03,Z 656.44,A -85,B 0,C 180,E1 17761.738,E2 17761.738} C_VEL
LIN {X 0,Y 355.042,Z 656.449,A -85,B 0,C 180,E1 17757.496,E2 17757.496} C_VEL
LIN {X 0,Y 355,Z 656.447,A -85,B 0,C 180,E1 17753.346,E2 17753.346} C_VEL
LIN {X 0,Y 354.984,Z 656.445,A -85,B 0,C 180,E1 17749.073,E2 17749.073} C_VEL
LIN {X 0,Y 355.013,Z 656.444,A -85,B 0,C 180,E1 17744.99,E2 17744.99} C_VEL
LIN {X 0,Y 355.03,Z 656.445,A -85,B 0,C 180,E1 17740.879,E2 17740.879} C_VEL
LIN {X 0,Y 355.013,Z 656.441,A -85,B 0,C 180,E1 17736.796,E2 17736.796} C_VEL
LIN {X 0,Y 354.966,Z 656.431,A -85,B 0,C 180,E1 17732.585,E2 17732.585} C_VEL
LIN {X 0,Y 355.002,Z 656.445,A -85,B 0,C 180,E1 17728.55,E2 17728.55} C_VEL
LIN {X 0,Y 355.026,Z 656.433,A -85,B 0,C 180,E1 17724.345,E2 17724.345} C_VEL
LIN {X 0,Y 355.019,Z 656.428,A -85,B 0,C 180,E1 17720.274,E2 17720.274} C_VEL
LIN {X 0,Y 354.975,Z 656.446,A -85,B 0,C 180,E1 17716.15,E2 17716.15} C_VEL
LIN {X 0,Y 354.993,Z 656.446,A -85,B 0,C 180,E1 17711.954,E2 17711.954} C_VEL
LIN {X 0,Y 355.02,Z 656.445,A -85,B 0,C 180,E1 17707.83,E2 17707.83} C_VEL
LIN {X 0,Y 355.031,Z 656.442,A -85,B 0,C 180,E1 17703.761,E2 17703.761} C_VEL
LIN {X 0,Y 354.996,Z 656.448,A -85,B 0,C 180,E1 17699.726,E2 17699.726} C_VEL
LIN {X 0,Y 354.979,Z 656.452,A -85,B 0,C 180,E1 17695.52,E2 17695.52} C_VEL
LIN {X 0,Y 355.03,Z 656.651,A -85,B 0,C 180,E1 17693.649,E2 17693.649} C_VEL
LIN {X 0,Y 363.675,Z 682.456,A -85,B 0,C 180,E1 17690.166,E2 17690.166} C_VEL
LIN {X 0,Y 370.671,Z 706.033,A -85,B 0,C 180,E1 17687.178,E2 17687.178} C_VEL
LIN {X 0,Y 373.356,Z 716.907,A -85,B 0,C 180,E1 17685.862,E2 17685.862} C_VEL
LIN {X 0,Y 370.453,Z 758.906,A -85,B 0,C 180,E1 17681.806,E2 17681.806} C_VEL
LIN {X 0,Y 367.521,Z 803.043,A -85,B 0,C 180,E1 17677.542,E2 17677.542} C_VEL
LIN {X 0,Y 366.739,Z 814.633,A -85,B 0,C 180,E1 17676.428,E2 17676.428} C_VEL
LIN {X 0,Y 365.372,Z 821.324,A -85,B 0,C 180,E1 17675.837,E2 17675.837} C_VEL
LIN {X 0,Y 358.275,Z 839.217,A -85,B 0,C 180,E1 17674.417,E2 17674.417} C_VEL
LIN {X 0,Y 357.238,Z 844.958,A -85,B 0,C 180,E1 17673.899,E2 17673.899} C_VEL
LIN {X 0,Y 356.558,Z 852.165,A -85,B 0,C 180,E1 17673.258,E2 17673.258} C_VEL
LIN {X 0,Y 352.163,Z 985.464,A -85,B 0,C 180,E1 17669.587,E2 17669.587} C_VEL
LIN {X 0,Y 351.814,Z 1004.869,A -85,B 0,C 180,E1 17668.918,E2 17668.918} C_VEL
LIN {X 0,Y 351.146,Z 1023.167,A -85,B 0,C 180,E1 17667.936,E2 17667.936} C_VEL
LIN {X 0,Y 350.354,Z 1039.55,A -85,B 0,C 180,E1 17666.718,E2 17666.718} C_VEL
LIN {X 0,Y 349.458,Z 1054.343,A -85,B 0,C 180,E1 17665.297,E2 17665.297} C_VEL
LIN {X 0,Y 348.463,Z 1069.137,A -85,B 0,C 180,E1 17663.502,E2 17663.502} C_VEL
LIN {X 0,Y 347.515,Z 1082.606,A -85,B 0,C 180,E1 17661.429,E2 17661.429} C_VEL
LIN {X 0,Y 346.806,Z 1093.352,A -85,B 0,C 180,E1 17659.359,E2 17659.359} C_VEL
LIN {X 0,Y 346.294,Z 1102.686,A -85,B 0,C 180,E1 17657.123,E2 17657.123} C_VEL
LIN {X 0,Y 346.011,Z 1110.446,A -85,B 0,C 180,E1 17654.728,E2 17654.728} C_VEL
LIN {X 0,Y 345.987,Z 1116.663,A -85,B 0,C 180,E1 17652.175,E2 17652.175} C_VEL
LIN {X 0,Y 346.292,Z 1121.053,A -85,B 0,C 180,E1 17649.469,E2 17649.469} C_VEL
LIN {X 0,Y 346.91,Z 1123.366,A -85,B 0,C 180,E1 17646.949,E2 17646.949} C_VEL
LIN {X 0,Y 347.961,Z 1123.889,A -85,B 0,C 180,E1 17644.281,E2 17644.281} C_VEL
LIN {X 0,Y 349.357,Z 1122.66,A -85,B 0,C 180,E1 17641.801,E2 17641.801} C_VEL
LIN {X 0,Y 351.312,Z 1119.391,A -85,B 0,C 180,E1 17639.181,E2 17639.181} C_VEL
LIN {X 0,Y 353.615,Z 1114.492,A -85,B 0,C 180,E1 17636.755,E2 17636.755} C_VEL
LIN {X 0,Y 356.352,Z 1107.501,A -85,B 0,C 180,E1 17634.361,E2 17634.361} C_VEL
LIN {X 0,Y 359.304,Z 1098.928,A -85,B 0,C 180,E1 17632.159,E2 17632.159} C_VEL
LIN {X 0,Y 362.351,Z 1088.823,A -85,B 0,C 180,E1 17630.146,E2 17630.146} C_VEL
LIN {X 0,Y 365.265,Z 1077.61,A -85,B 0,C 180,E1 17628.39,E2 17628.39} C_VEL
LIN {X 0,Y 368.335,Z 1063.693,A -85,B 0,C 180,E1 17626.656,E2 17626.656} C_VEL
LIN {X 0,Y 370.994,Z 1049.166,A -85,B 0,C 180,E1 17625.241,E2 17625.241} C_VEL
LIN {X 0,Y 372.958,Z 1035.359,A -85,B 0,C 180,E1 17624.207,E2 17624.207} C_VEL
LIN {X 0,Y 374.701,Z 1019.719,A -85,B 0,C 180,E1 17623.287,E2 17623.287} C_VEL
LIN {X 0,Y 375.987,Z 1001.001,A -85,B 0,C 180,E1 17622.514,E2 17622.514} C_VEL
LIN {X 0,Y 379.61,Z 956.712,A -85,B 0,C 180,E1 17621.113,E2 17621.113} C_VEL
LIN {X 0,Y 388.204,Z 871.758,A -85,B 0,C 180,E1 17618.553,E2 17618.553} C_VEL
LIN {X 0,Y 388.587,Z 867.556,A -85,B 0,C 180,E1 17618.169,E2 17618.169} C_VEL
LIN {X 0,Y 396.044,Z 823.613,A -85,B 0,C 180,E1 17613.696,E2 17613.696} C_VEL
LIN {X 0,Y 405.294,Z 778.073,A -85,B 0,C 180,E1 17609.041,E2 17609.041} C_VEL
LIN {X 0,Y 409.542,Z 759.498,A -85,B 0,C 180,E1 17607.121,E2 17607.121} C_VEL
LIN {X 0,Y 408.898,Z 752.199,A -85,B 0,C 180,E1 17605.243,E2 17605.243} C_VEL
LIN {X 0,Y 408.3,Z 746.884,A -85,B 0,C 180,E1 17603.436,E2 17603.436} C_VEL
LIN {X 0,Y 407.785,Z 742.218,A -85,B 0,C 180,E1 17601.296,E2 17601.296} C_VEL
LIN {X 0,Y 407.516,Z 741.036,A -85,B 0,C 180,E1 17600.224,E2 17600.224} C_VEL
LIN {X 0,Y 401.052,Z 755.903,A -85,B 0,C 180,E1 17597.344,E2 17597.344} C_VEL
LIN {X 0,Y 399.069,Z 762.565,A -85,B 0,C 180,E1 17596.118,E2 17596.118} C_VEL
LIN {X 0,Y 382.129,Z 977.263,A -85,B 0,C 180,E1 17590.722,E2 17590.722} C_VEL
LIN {X 0,Y 379.337,Z 1001.785,A -85,B 0,C 180,E1 17589.827,E2 17589.827} C_VEL
LIN {X 0,Y 376.012,Z 1025.377,A -85,B 0,C 180,E1 17588.672,E2 17588.672} C_VEL
LIN {X 0,Y 372.563,Z 1046.842,A -85,B 0,C 180,E1 17587.337,E2 17587.337} C_VEL
LIN {X 0,Y 368.821,Z 1067.738,A -85,B 0,C 180,E1 17585.745,E2 17585.745} C_VEL
LIN {X 0,Y 364.891,Z 1088.154,A -85,B 0,C 180,E1 17583.867,E2 17583.867} C_VEL
LIN {X 0,Y 361.014,Z 1107.399,A -85,B 0,C 180,E1 17581.748,E2 17581.748} C_VEL
LIN {X 0,Y 357.192,Z 1125.807,A -85,B 0,C 180,E1 17579.33,E2 17579.33} C_VEL
LIN {X 0,Y 353.728,Z 1142.517,A -85,B 0,C 180,E1 17576.705,E2 17576.705} C_VEL
LIN {X 0,Y 350.881,Z 1156.866,A -85,B 0,C 180,E1 17574.045,E2 17574.045} C_VEL
LIN {X 0,Y 348.458,Z 1170.118,A -85,B 0,C 180,E1 17571.153,E2 17571.153} C_VEL
LIN {X 0,Y 346.614,Z 1181.69,A -85,B 0,C 180,E1 17568.15,E2 17568.15} C_VEL
LIN {X 0,Y 345.356,Z 1191.366,A -85,B 0,C 180,E1 17565.101,E2 17565.101} C_VEL
LIN {X 0,Y 344.576,Z 1200.124,A -85,B 0,C 180,E1 17561.717,E2 17561.717} C_VEL
LIN {X 0,Y 344.305,Z 1206.649,A -85,B 0,C 180,E1 17558.515,E2 17558.515} C_VEL
LIN {X 0,Y 344.289,Z 1211.334,A -85,B 0,C 180,E1 17555.33,E2 17555.33} C_VEL
LIN {X 0,Y 344.336,Z 1214.505,A -85,B 0,C 180,E1 17552.161,E2 17552.161} C_VEL
LIN {X 0,Y 344.29,Z 1216.01,A -85,B 0,C 180,E1 17549.166,E2 17549.166} C_VEL
LIN {X 0,Y 344.138,Z 1216.215,A -85,B 0,C 180,E1 17545.999,E2 17545.999} C_VEL
LIN {X 0,Y 344.062,Z 1214.881,A -85,B 0,C 180,E1 17542.819,E2 17542.819} C_VEL
LIN {X 0,Y 344.319,Z 1211.846,A -85,B 0,C 180,E1 17539.287,E2 17539.287} C_VEL
LIN {X 0,Y 345.24,Z 1207.138,A -85,B 0,C 180,E1 17535.746,E2 17535.746} C_VEL
LIN {X 0,Y 347.025,Z 1200.69,A -85,B 0,C 180,E1 17532.215,E2 17532.215} C_VEL
LIN {X 0,Y 350.002,Z 1192.148,A -85,B 0,C 180,E1 17528.549,E2 17528.549} C_VEL
LIN {X 0,Y 354.246,Z 1181.689,A -85,B 0,C 180,E1 17524.949,E2 17524.949} C_VEL
LIN {X 0,Y 359.912,Z 1168.943,A -85,B 0,C 180,E1 17521.394,E2 17521.394} C_VEL
LIN {X 0,Y 366.818,Z 1154.509,A -85,B 0,C 180,E1 17518.073,E2 17518.073} C_VEL
LIN {X 0,Y 375.303,Z 1137.701,A -85,B 0,C 180,E1 17514.866,E2 17514.866} C_VEL
LIN {X 0,Y 385.36,Z 1118.626,A -85,B 0,C 180,E1 17511.862,E2 17511.862} C_VEL
LIN {X 0,Y 396.484,Z 1098.227,A -85,B 0,C 180,E1 17509.217,E2 17509.217} C_VEL
LIN {X 0,Y 408.254,Z 1077.195,A -85,B 0,C 180,E1 17506.991,E2 17506.991} C_VEL
LIN {X 0,Y 420.424,Z 1055.677,A -85,B 0,C 180,E1 17505.156,E2 17505.156} C_VEL
LIN {X 0,Y 427.645,Z 1042.715,A -85,B 0,C 180,E1 17504.217,E2 17504.217} C_VEL
LIN {X 0,Y 415.532,Z 1063.319,A -85,B 0,C 180,E1 17502.361,E2 17502.361} C_VEL
LIN {X 0,Y 403.584,Z 1083.361,A -85,B 0,C 180,E1 17500.105,E2 17500.105} C_VEL
LIN {X 0,Y 392.421,Z 1102.048,A -85,B 0,C 180,E1 17497.518,E2 17497.518} C_VEL
LIN {X 0,Y 382.15,Z 1119.278,A -85,B 0,C 180,E1 17494.598,E2 17494.598} C_VEL
LIN {X 0,Y 373.271,Z 1134.244,A -85,B 0,C 180,E1 17491.493,E2 17491.493} C_VEL
LIN {X 0,Y 365.705,Z 1147.051,A -85,B 0,C 180,E1 17488.233,E2 17488.233} C_VEL
LIN {X 0,Y 359.685,Z 1157.383,A -85,B 0,C 180,E1 17484.999,E2 17484.999} C_VEL
LIN {X 0,Y 354.518,Z 1166.506,A -85,B 0,C 180,E1 17481.446,E2 17481.446} C_VEL
LIN {X 0,Y 350.529,Z 1173.809,A -85,B 0,C 180,E1 17477.775,E2 17477.775} C_VEL
LIN {X 0,Y 347.765,Z 1179.151,A -85,B 0,C 180,E1 17474.149,E2 17474.149} C_VEL
LIN {X 0,Y 345.931,Z 1182.668,A -85,B 0,C 180,E1 17470.495,E2 17470.495} C_VEL
LIN {X 0,Y 344.921,Z 1184.461,A -85,B 0,C 180,E1 17466.997,E2 17466.997} C_VEL
LIN {X 0,Y 344.44,Z 1184.79,A -85,B 0,C 180,E1 17463.665,E2 17463.665} C_VEL
LIN {X 0,Y 344.225,Z 1183.528,A -85,B 0,C 180,E1 17460.336,E2 17460.336} C_VEL
LIN {X 0,Y 344.184,Z 1180.802,A -85,B 0,C 180,E1 17456.961,E2 17456.961} C_VEL
LIN {X 0,Y 344.289,Z 1176.832,A -85,B 0,C 180,E1 17453.835,E2 17453.835} C_VEL
LIN {X 0,Y 344.66,Z 1170.955,A -85,B 0,C 180,E1 17450.486,E2 17450.486} C_VEL
LIN {X 0,Y 345.392,Z 1163.779,A -85,B 0,C 180,E1 17447.294,E2 17447.294} C_VEL
LIN {X 0,Y 346.609,Z 1154.763,A -85,B 0,C 180,E1 17444.098,E2 17444.098} C_VEL
LIN {X 0,Y 348.416,Z 1143.8,A -85,B 0,C 180,E1 17440.908,E2 17440.908} C_VEL
LIN {X 0,Y 350.888,Z 1130.661,A -85,B 0,C 180,E1 17437.733,E2 17437.733} C_VEL
LIN {X 0,Y 353.698,Z 1116.784,A -85,B 0,C 180,E1 17434.914,E2 17434.914} C_VEL
LIN {X 0,Y 357.012,Z 1101.015,A -85,B 0,C 180,E1 17432.209,E2 17432.209} C_VEL
LIN {X 0,Y 360.636,Z 1083.607,A -85,B 0,C 180,E1 17429.699,E2 17429.699} C_VEL
LIN {X 0,Y 364.376,Z 1065.268,A -85,B 0,C 180,E1 17427.468,E2 17427.468} C_VEL
LIN {X 0,Y 368.339,Z 1044.751,A -85,B 0,C 180,E1 17425.371,E2 17425.371} C_VEL
LIN {X 0,Y 372.129,Z 1023.598,A -85,B 0,C 180,E1 17423.577,E2 17423.577} C_VEL
LIN {X 0,Y 375.449,Z 1003.095,A -85,B 0,C 180,E1 17422.136,E2 17422.136} C_VEL
LIN {X 0,Y 378.797,Z 979.299,A -85,B 0,C 180,E1 17420.793,E2 17420.793} C_VEL
LIN {X 0,Y 381.647,Z 954.66,A -85,B 0,C 180,E1 17419.725,E2 17419.725} C_VEL
LIN {X 0,Y 383.778,Z 930.583,A -85,B 0,C 180,E1 17418.968,E2 17418.968} C_VEL
LIN {X 0,Y 398.115,Z 745.601,A -85,B 0,C 180,E1 17414.369,E2 17414.369} C_VEL
LIN {X 0,Y 380.743,Z 714.315,A -85,B 0,C 180,E1 17411.464,E2 17411.464} C_VEL
LIN {X 0,Y 365.292,Z 688.06,A -85,B 0,C 180,E1 17408.642,E2 17408.642} C_VEL
LIN {X 0,Y 351.852,Z 666.276,A -85,B 0,C 180,E1 17405.985,E2 17405.985} C_VEL
LIN {X 0,Y 349.24,Z 662,A -85,B 0,C 180,E1 17405.436,E2 17405.436} C_VEL
LIN {X 0,Y 347.35,Z 658.799,A -85,B 0,C 180,E1 17405.026,E2 17405.026} C_VEL
LIN {X 0,Y 347.06,Z 657.429,A -85,B 0,C 180,E1 17404.884,E2 17404.884} C_VEL
LIN {X 0,Y 347.096,Z 657.434,A -85,B 0,C 180,E1 17400.658,E2 17400.658} C_VEL
LIN {X 0,Y 347.065,Z 657.43,A -85,B 0,C 180,E1 17396.34,E2 17396.34} C_VEL
LIN {X 0,Y 347.026,Z 657.432,A -85,B 0,C 180,E1 17392.178,E2 17392.178} C_VEL
LIN {X 0,Y 347.066,Z 657.424,A -85,B 0,C 180,E1 17387.957,E2 17387.957} C_VEL
LIN {X 0,Y 347.095,Z 657.416,A -85,B 0,C 180,E1 17383.836,E2 17383.836} C_VEL
LIN {X 0,Y 347.077,Z 657.427,A -85,B 0,C 180,E1 17379.621,E2 17379.621} C_VEL
LIN {X 0,Y 347.051,Z 657.44,A -85,B 0,C 180,E1 17375.458,E2 17375.458} C_VEL
LIN {X 0,Y 347.069,Z 657.426,A -85,B 0,C 180,E1 17370.993,E2 17370.993} C_VEL
LIN {X 0,Y 347.083,Z 657.414,A -85,B 0,C 180,E1 17366.865,E2 17366.865} C_VEL
LIN {X 0,Y 347.102,Z 657.431,A -85,B 0,C 180,E1 17362.554,E2 17362.554} C_VEL
LIN {X 0,Y 347.065,Z 657.407,A -85,B 0,C 180,E1 17358.365,E2 17358.365} C_VEL
LIN {X 0,Y 347.04,Z 657.437,A -85,B 0,C 180,E1 17354.117,E2 17354.117} C_VEL
LIN {X 0,Y 347.069,Z 657.432,A -85,B 0,C 180,E1 17349.902,E2 17349.902} C_VEL
LIN {X 0,Y 347.09,Z 657.432,A -85,B 0,C 180,E1 17345.675,E2 17345.675} C_VEL
LIN {X 0,Y 347.061,Z 657.436,A -85,B 0,C 180,E1 17341.432,E2 17341.432} C_VEL
LIN {X 0,Y 347.023,Z 657.443,A -85,B 0,C 180,E1 17337.204,E2 17337.204} C_VEL
LIN {X 0,Y 347.092,Z 657.586,A -85,B 0,C 180,E1 17334.266,E2 17334.266} C_VEL
LIN {X 0,Y 355.815,Z 683.532,A -85,B 0,C 180,E1 17330.681,E2 17330.681} C_VEL
LIN {X 0,Y 363.098,Z 707.952,A -85,B 0,C 180,E1 17327.556,E2 17327.556} C_VEL
LIN {X 0,Y 365.845,Z 719.2,A -85,B 0,C 180,E1 17326.175,E2 17326.175} C_VEL
LIN {X 0,Y 362.788,Z 761.381,A -85,B 0,C 180,E1 17322.041,E2 17322.041} C_VEL
LIN {X 0,Y 359.739,Z 805.964,A -85,B 0,C 180,E1 17317.692,E2 17317.692} C_VEL
LIN {X 0,Y 357.238,Z 844.958,A -85,B 0,C 180,E1 17313.899,E2 17313.899} C_VEL
LIN {X 0,Y 356.401,Z 849.878,A -85,B 0,C 180,E1 17313.535,E2 17313.535} C_VEL
LIN {X 0,Y 353.942,Z 857.055,A -85,B 0,C 180,E1 17313.26,E2 17313.26} C_VEL
LIN {X 0,Y 348.948,Z 870.828,A -85,B 0,C 180,E1 17313.025,E2 17313.025} C_VEL
LIN {X 0,Y 347.731,Z 878.564,A -85,B 0,C 180,E1 17312.843,E2 17312.843} C_VEL
LIN {X 0,Y 344.248,Z 987.113,A -85,B 0,C 180,E1 17309.755,E2 17309.755} C_VEL
LIN {X 0,Y 343.876,Z 1006.079,A -85,B 0,C 180,E1 17309.07,E2 17309.07} C_VEL
LIN {X 0,Y 343.182,Z 1024.353,A -85,B 0,C 180,E1 17308.055,E2 17308.055} C_VEL
LIN {X 0,Y 342.318,Z 1041.555,A -85,B 0,C 180,E1 17306.728,E2 17306.728} C_VEL
LIN {X 0,Y 341.376,Z 1056.582,A -85,B 0,C 180,E1 17305.22,E2 17305.22} C_VEL
LIN {X 0,Y 340.433,Z 1070.361,A -85,B 0,C 180,E1 17303.493,E2 17303.493} C_VEL
LIN {X 0,Y 339.497,Z 1083.557,A -85,B 0,C 180,E1 17301.416,E2 17301.416} C_VEL
LIN {X 0,Y 338.786,Z 1094.332,A -85,B 0,C 180,E1 17299.298,E2 17299.298} C_VEL
LIN {X 0,Y 338.282,Z 1103.695,A -85,B 0,C 180,E1 17297.011,E2 17297.011} C_VEL
LIN {X 0,Y 338.012,Z 1111.48,A -85,B 0,C 180,E1 17294.559,E2 17294.559} C_VEL
LIN {X 0,Y 338.02,Z 1117.687,A -85,B 0,C 180,E1 17291.946,E2 17291.946} C_VEL
LIN {X 0,Y 338.375,Z 1122.098,A -85,B 0,C 180,E1 17289.178,E2 17289.178} C_VEL
LIN {X 0,Y 339.065,Z 1124.445,A -85,B 0,C 180,E1 17286.6,E2 17286.6} C_VEL
LIN {X 0,Y 340.217,Z 1124.992,A -85,B 0,C 180,E1 17283.872,E2 17283.872} C_VEL
LIN {X 0,Y 341.743,Z 1123.807,A -85,B 0,C 180,E1 17281.338,E2 17281.338} C_VEL
LIN {X 0,Y 343.86,Z 1120.575,A -85,B 0,C 180,E1 17278.663,E2 17278.663} C_VEL
LIN {X 0,Y 346.331,Z 1115.688,A -85,B 0,C 180,E1 17276.189,E2 17276.189} C_VEL
LIN {X 0,Y 349.271,Z 1108.78,A -85,B 0,C 180,E1 17273.751,E2 17273.751} C_VEL
LIN {X 0,Y 352.189,Z 1100.978,A -85,B 0,C 180,E1 17271.671,E2 17271.671} C_VEL
LIN {X 0,Y 355.382,Z 1091.02,A -85,B 0,C 180,E1 17269.623,E2 17269.623} C_VEL
LIN {X 0,Y 358.621,Z 1079.662,A -85,B 0,C 180,E1 17267.763,E2 17267.763} C_VEL
LIN {X 0,Y 361.881,Z 1066.049,A -85,B 0,C 180,E1 17266.006,E2 17266.006} C_VEL
LIN {X 0,Y 364.665,Z 1051.745,A -85,B 0,C 180,E1 17264.572,E2 17264.572} C_VEL
LIN {X 0,Y 366.759,Z 1038.426,A -85,B 0,C 180,E1 17263.526,E2 17263.526} C_VEL
LIN {X 0,Y 368.399,Z 1025.467,A -85,B 0,C 180,E1 17262.707,E2 17262.707} C_VEL
LIN {X 0,Y 369.822,Z 1009.897,A -85,B 0,C 180,E1 17261.953,E2 17261.953} C_VEL
LIN {X 0,Y 372.869,Z 971.378,A -85,B 0,C 180,E1 17260.642,E2 17260.642} C_VEL
LIN {X 0,Y 383.273,Z 873.705,A -85,B 0,C 180,E1 17257.649,E2 17257.649} C_VEL
LIN {X 0,Y 383.387,Z 870.734,A -85,B 0,C 180,E1 17257.398,E2 17257.398} C_VEL
LIN {X 0,Y 391.697,Z 825.411,A -85,B 0,C 180,E1 17252.725,E2 17252.725} C_VEL
LIN {X 0,Y 401.738,Z 779.502,A -85,B 0,C 180,E1 17247.982,E2 17247.982} C_VEL
LIN {X 0,Y 405.471,Z 764.356,A -85,B 0,C 180,E1 17246.382,E2 17246.382} C_VEL
LIN {X 0,Y 405.01,Z 757.073,A -85,B 0,C 180,E1 17244.361,E2 17244.361} C_VEL
LIN {X 0,Y 404.635,Z 751.544,A -85,B 0,C 180,E1 17242.203,E2 17242.203} C_VEL
LIN {X 0,Y 404.436,Z 748.736,A -85,B 0,C 180,E1 17240.566,E2 17240.566} C_VEL
LIN {X 0,Y 397.737,Z 763.891,A -85,B 0,C 180,E1 17237.641,E2 17237.641} C_VEL
LIN {X 0,Y 396.82,Z 766.529,A -85,B 0,C 180,E1 17237.155,E2 17237.155} C_VEL
LIN {X 0,Y 392.265,Z 778.609,A -85,B 0,C 180,E1 17236.587,E2 17236.587} C_VEL
LIN {X 0,Y 390.588,Z 784.107,A -85,B 0,C 180,E1 17236.249,E2 17236.249} C_VEL
LIN {X 0,Y 375.038,Z 976.533,A -85,B 0,C 180,E1 17231.286,E2 17231.286} C_VEL
LIN {X 0,Y 372.138,Z 1001.391,A -85,B 0,C 180,E1 17230.359,E2 17230.359} C_VEL
LIN {X 0,Y 368.725,Z 1024.971,A -85,B 0,C 180,E1 17229.182,E2 17229.182} C_VEL
LIN {X 0,Y 365.2,Z 1046.394,A -85,B 0,C 180,E1 17227.825,E2 17227.825} C_VEL
LIN {X 0,Y 361.199,Z 1068.201,A -85,B 0,C 180,E1 17226.128,E2 17226.128} C_VEL
LIN {X 0,Y 356.92,Z 1089.822,A -85,B 0,C 180,E1 17224.072,E2 17224.072} C_VEL
LIN {X 0,Y 352.958,Z 1108.901,A -85,B 0,C 180,E1 17221.89,E2 17221.89} C_VEL
LIN {X 0,Y 349.201,Z 1126.629,A -85,B 0,C 180,E1 17219.482,E2 17219.482} C_VEL
LIN {X 0,Y 345.612,Z 1143.622,A -85,B 0,C 180,E1 17216.733,E2 17216.733} C_VEL
LIN {X 0,Y 342.673,Z 1158.162,A -85,B 0,C 180,E1 17213.925,E2 17213.925} C_VEL
LIN {X 0,Y 340.177,Z 1171.672,A -85,B 0,C 180,E1 17210.831,E2 17210.831} C_VEL
LIN {X 0,Y 338.385,Z 1183.043,A -85,B 0,C 180,E1 17207.717,E2 17207.717} C_VEL
LIN {X 0,Y 337.158,Z 1192.987,A -85,B 0,C 180,E1 17204.422,E2 17204.422} C_VEL
LIN {X 0,Y 336.52,Z 1200.883,A -85,B 0,C 180,E1 17201.133,E2 17201.133} C_VEL
LIN {X 0,Y 336.302,Z 1207.325,A -85,B 0,C 180,E1 17197.686,E2 17197.686} C_VEL
LIN {X 0,Y 336.322,Z 1211.554,A -85,B 0,C 180,E1 17194.602,E2 17194.602} C_VEL
LIN {X 0,Y 336.359,Z 1214.376,A -85,B 0,C 180,E1 17191.36,E2 17191.36} C_VEL
LIN {X 0,Y 336.278,Z 1215.64,A -85,B 0,C 180,E1 17188.464,E2 17188.464} C_VEL
LIN {X 0,Y 336.099,Z 1215.563,A -85,B 0,C 180,E1 17185.048,E2 17185.048} C_VEL
LIN {X 0,Y 336.082,Z 1214.056,A -85,B 0,C 180,E1 17181.788,E2 17181.788} C_VEL
LIN {X 0,Y 336.528,Z 1210.734,A -85,B 0,C 180,E1 17178.168,E2 17178.168} C_VEL
LIN {X 0,Y 337.736,Z 1205.849,A -85,B 0,C 180,E1 17174.545,E2 17174.545} C_VEL
LIN {X 0,Y 340.039,Z 1198.852,A -85,B 0,C 180,E1 17170.769,E2 17170.769} C_VEL
LIN {X 0,Y 343.558,Z 1190.027,A -85,B 0,C 180,E1 17167.044,E2 17167.044} C_VEL
LIN {X 0,Y 348.428,Z 1179.354,A -85,B 0,C 180,E1 17163.403,E2 17163.403} C_VEL
LIN {X 0,Y 354.719,Z 1166.753,A -85,B 0,C 180,E1 17159.882,E2 17159.882} C_VEL
LIN {X 0,Y 362.875,Z 1151.389,A -85,B 0,C 180,E1 17156.367,E2 17156.367} C_VEL
LIN {X 0,Y 372.526,Z 1134.109,A -85,B 0,C 180,E1 17153.12,E2 17153.12} C_VEL
LIN {X 0,Y 383.221,Z 1115.697,A -85,B 0,C 180,E1 17150.262,E2 17150.262} C_VEL
LIN {X 0,Y 395.578,Z 1095.161,A -85,B 0,C 180,E1 17147.651,E2 17147.651} C_VEL
LIN {X 0,Y 408.25,Z 1074.569,A -85,B 0,C 180,E1 17145.533,E2 17145.533} C_VEL
LIN {X 0,Y 418.425,Z 1058.134,A -85,B 0,C 180,E1 17144.128,E2 17144.128} C_VEL
LIN {X 0,Y 406.345,Z 1076.701,A -85,B 0,C 180,E1 17142.207,E2 17142.207} C_VEL
LIN {X 0,Y 393.885,Z 1095.683,A -85,B 0,C 180,E1 17139.773,E2 17139.773} C_VEL
LIN {X 0,Y 382.322,Z 1113.33,A -85,B 0,C 180,E1 17136.982,E2 17136.982} C_VEL
LIN {X 0,Y 372.211,Z 1128.858,A -85,B 0,C 180,E1 17133.973,E2 17133.973} C_VEL
LIN {X 0,Y 363.507,Z 1142.373,A -85,B 0,C 180,E1 17130.775,E2 17130.775} C_VEL
LIN {X 0,Y 355.824,Z 1154.36,A -85,B 0,C 180,E1 17127.264,E2 17127.264} C_VEL
LIN {X 0,Y 349.568,Z 1164.273,A -85,B 0,C 180,E1 17123.61,E2 17123.61} C_VEL
LIN {X 0,Y 344.867,Z 1171.904,A -85,B 0,C 180,E1 17120.01,E2 17120.01} C_VEL
LIN {X 0,Y 341.23,Z 1178.028,A -85,B 0,C 180,E1 17116.167,E2 17116.167} C_VEL
LIN {X 0,Y 338.85,Z 1182.178,A -85,B 0,C 180,E1 17112.443,E2 17112.443} C_VEL
LIN {X 0,Y 337.371,Z 1184.608,A -85,B 0,C 180,E1 17108.697,E2 17108.697} C_VEL
LIN {X 0,Y 336.614,Z 1185.3,A -85,B 0,C 180,E1 17105.116,E2 17105.116} C_VEL
LIN {X 0,Y 336.292,Z 1184.472,A -85,B 0,C 180,E1 17101.537,E2 17101.537} C_VEL
LIN {X 0,Y 336.184,Z 1182.278,A -85,B 0,C 180,E1 17098.299,E2 17098.299} C_VEL
LIN {X 0,Y 336.233,Z 1178.474,A -85,B 0,C 180,E1 17094.885,E2 17094.885} C_VEL
LIN {X 0,Y 336.498,Z 1173.403,A -85,B 0,C 180,E1 17091.632,E2 17091.632} C_VEL
LIN {X 0,Y 337.095,Z 1166.636,A -85,B 0,C 180,E1 17088.368,E2 17088.368} C_VEL
LIN {X 0,Y 338.225,Z 1157.719,A -85,B 0,C 180,E1 17084.925,E2 17084.925} C_VEL
LIN {X 0,Y 339.9,Z 1147.347,A -85,B 0,C 180,E1 17081.658,E2 17081.658} C_VEL
LIN {X 0,Y 342.096,Z 1135.498,A -85,B 0,C 180,E1 17078.575,E2 17078.575} C_VEL
LIN {X 0,Y 344.757,Z 1122.285,A -85,B 0,C 180,E1 17075.684,E2 17075.684} C_VEL
LIN {X 0,Y 348.138,Z 1106.339,A -85,B 0,C 180,E1 17072.74,E2 17072.74} C_VEL
LIN {X 0,Y 351.697,Z 1089.831,A -85,B 0,C 180,E1 17070.168,E2 17070.168} C_VEL
LIN {X 0,Y 355.505,Z 1071.847,A -85,B 0,C 180,E1 17067.797,E2 17067.797} C_VEL
LIN {X 0,Y 359.483,Z 1052.151,A -85,B 0,C 180,E1 17065.628,E2 17065.628} C_VEL
LIN {X 0,Y 363.343,Z 1031.535,A -85,B 0,C 180,E1 17063.73,E2 17063.73} C_VEL
LIN {X 0,Y 367.025,Z 1010.132,A -85,B 0,C 180,E1 17062.102,E2 17062.102} C_VEL
LIN {X 0,Y 370.477,Z 987.297,A -85,B 0,C 180,E1 17060.691,E2 17060.691} C_VEL
LIN {X 0,Y 373.412,Z 964.322,A -85,B 0,C 180,E1 17059.568,E2 17059.568} C_VEL
LIN {X 0,Y 375.903,Z 940.547,A -85,B 0,C 180,E1 17058.69,E2 17058.69} C_VEL
LIN {X 0,Y 391.287,Z 748.41,A -85,B 0,C 180,E1 17053.78,E2 17053.78} C_VEL
LIN {X 0,Y 374.098,Z 717.249,A -85,B 0,C 180,E1 17050.808,E2 17050.808} C_VEL
LIN {X 0,Y 357.065,Z 688.387,A -85,B 0,C 180,E1 17047.6,E2 17047.6} C_VEL
LIN {X 0,Y 343.991,Z 667.324,A -85,B 0,C 180,E1 17044.91,E2 17044.91} C_VEL
LIN {X 0,Y 341.371,Z 663.028,A -85,B 0,C 180,E1 17044.334,E2 17044.334} C_VEL
LIN {X 0,Y 339.449,Z 659.817,A -85,B 0,C 180,E1 17043.908,E2 17043.908} C_VEL
LIN {X 0,Y 339.144,Z 658.424,A -85,B 0,C 180,E1 17043.764,E2 17043.764} C_VEL
LIN {X 0,Y 339.159,Z 658.414,A -85,B 0,C 180,E1 17039.497,E2 17039.497} C_VEL
LIN {X 0,Y 339.138,Z 658.419,A -85,B 0,C 180,E1 17035.312,E2 17035.312} C_VEL
LIN {X 0,Y 339.093,Z 658.428,A -85,B 0,C 180,E1 17031.087,E2 17031.087} C_VEL
LIN {X 0,Y 339.121,Z 658.422,A -85,B 0,C 180,E1 17026.797,E2 17026.797} C_VEL
LIN {X 0,Y 339.147,Z 658.411,A -85,B 0,C 180,E1 17022.604,E2 17022.604} C_VEL
LIN {X 0,Y 339.123,Z 658.408,A -85,B 0,C 180,E1 17018.309,E2 17018.309} C_VEL
LIN {X 0,Y 339.082,Z 658.424,A -85,B 0,C 180,E1 17014.061,E2 17014.061} C_VEL
LIN {X 0,Y 339.119,Z 658.427,A -85,B 0,C 180,E1 17009.664,E2 17009.664} C_VEL
LIN {X 0,Y 339.147,Z 658.399,A -85,B 0,C 180,E1 17005.437,E2 17005.437} C_VEL
LIN {X 0,Y 339.133,Z 658.419,A -85,B 0,C 180,E1 17001.183,E2 17001.183} C_VEL
LIN {X 0,Y 339.11,Z 658.413,A -85,B 0,C 180,E1 16996.88,E2 16996.88} C_VEL
LIN {X 0,Y 339.133,Z 658.42,A -85,B 0,C 180,E1 16992.501,E2 16992.501} C_VEL
LIN {X 0,Y 339.15,Z 658.421,A -85,B 0,C 180,E1 16988.196,E2 16988.196} C_VEL
LIN {X 0,Y 339.157,Z 658.418,A -85,B 0,C 180,E1 16983.945,E2 16983.945} C_VEL
LIN {X 0,Y 339.118,Z 658.426,A -85,B 0,C 180,E1 16979.725,E2 16979.725} C_VEL
LIN {X 0,Y 339.098,Z 658.43,A -85,B 0,C 180,E1 16975.316,E2 16975.316} C_VEL
LIN {X 0,Y 339.105,Z 658.462,A -85,B 0,C 180,E1 16974.905,E2 16974.905} C_VEL
LIN {X 0,Y 347.632,Z 683.491,A -85,B 0,C 180,E1 16971.383,E2 16971.383} C_VEL
LIN {X 0,Y 354.671,Z 706.909,A -85,B 0,C 180,E1 16968.296,E2 16968.296} C_VEL
LIN {X 0,Y 358.332,Z 721.383,A -85,B 0,C 180,E1 16966.504,E2 16966.504} C_VEL
LIN {X 0,Y 355.188,Z 763.426,A -85,B 0,C 180,E1 16962.342,E2 16962.342} C_VEL
LIN {X 0,Y 352.019,Z 807.89,A -85,B 0,C 180,E1 16957.943,E2 16957.943} C_VEL
LIN {X 0,Y 349.257,Z 849.504,A -85,B 0,C 180,E1 16953.843,E2 16953.843} C_VEL
LIN {X 0,Y 348.784,Z 853.001,A -85,B 0,C 180,E1 16953.563,E2 16953.563} C_VEL
LIN {X 0,Y 347.731,Z 878.564,A -85,B 0,C 180,E1 16952.843,E2 16952.843} C_VEL
LIN {X 0,Y 346.44,Z 886.151,A -85,B 0,C 180,E1 16952.669,E2 16952.669} C_VEL
LIN {X 0,Y 339.558,Z 906.151,A -85,B 0,C 180,E1 16952.324,E2 16952.324} C_VEL
LIN {X 0,Y 338.603,Z 912.667,A -85,B 0,C 180,E1 16952.158,E2 16952.158} C_VEL
LIN {X 0,Y 336.26,Z 992.386,A -85,B 0,C 180,E1 16949.8,E2 16949.8} C_VEL
LIN {X 0,Y 335.833,Z 1010.098,A -85,B 0,C 180,E1 16949.076,E2 16949.076} C_VEL
LIN {X 0,Y 335.176,Z 1026.33,A -85,B 0,C 180,E1 16948.117,E2 16948.117} C_VEL
LIN {X 0,Y 334.286,Z 1043.42,A -85,B 0,C 180,E1 16946.749,E2 16946.749} C_VEL
LIN {X 0,Y 333.277,Z 1059.035,A -85,B 0,C 180,E1 16945.116,E2 16945.116} C_VEL
LIN {X 0,Y 332.358,Z 1072.184,A -85,B 0,C 180,E1 16943.394,E2 16943.394} C_VEL
LIN {X 0,Y 331.445,Z 1085.025,A -85,B 0,C 180,E1 16941.312,E2 16941.312} C_VEL
LIN {X 0,Y 330.718,Z 1096.088,A -85,B 0,C 180,E1 16939.054,E2 16939.054} C_VEL
LIN {X 0,Y 330.241,Z 1105.272,A -85,B 0,C 180,E1 16936.712,E2 16936.712} C_VEL
LIN {X 0,Y 329.997,Z 1113.399,A -85,B 0,C 180,E1 16934.024,E2 16934.024} C_VEL
LIN {X 0,Y 330.069,Z 1119.013,A -85,B 0,C 180,E1 16931.529,E2 16931.529} C_VEL
LIN {X 0,Y 330.505,Z 1123.372,A -85,B 0,C 180,E1 16928.696,E2 16928.696} C_VEL
LIN {X 0,Y 331.295,Z 1125.602,A -85,B 0,C 180,E1 16926.06,E2 16926.06} C_VEL
LIN {X 0,Y 332.594,Z 1126.098,A -85,B 0,C 180,E1 16923.271,E2 16923.271} C_VEL
LIN {X 0,Y 334.282,Z 1124.815,A -85,B 0,C 180,E1 16920.682,E2 16920.682} C_VEL
LIN {X 0,Y 336.605,Z 1121.508,A -85,B 0,C 180,E1 16917.954,E2 16917.954} C_VEL
LIN {X 0,Y 339.298,Z 1116.567,A -85,B 0,C 180,E1 16915.433,E2 16915.433} C_VEL
LIN {X 0,Y 342.474,Z 1109.58,A -85,B 0,C 180,E1 16912.953,E2 16912.953} C_VEL
LIN {X 0,Y 345.843,Z 1100.947,A -85,B 0,C 180,E1 16910.679,E2 16910.679} C_VEL
LIN {X 0,Y 349.329,Z 1090.864,A -85,B 0,C 180,E1 16908.606,E2 16908.606} C_VEL
LIN {X 0,Y 352.773,Z 1079.108,A -85,B 0,C 180,E1 16906.724,E2 16906.724} C_VEL
LIN {X 0,Y 356.087,Z 1065.727,A -85,B 0,C 180,E1 16905.025,E2 16905.025} C_VEL
LIN {X 0,Y 359.092,Z 1051.25,A -85,B 0,C 180,E1 16903.58,E2 16903.58} C_VEL
LIN {X 0,Y 361.826,Z 1034.433,A -85,B 0,C 180,E1 16902.3,E2 16902.3} C_VEL
LIN {X 0,Y 363.89,Z 1016.353,A -85,B 0,C 180,E1 16901.296,E2 16901.296} C_VEL
LIN {X 0,Y 366.34,Z 985.472,A -85,B 0,C 180,E1 16900.147,E2 16900.147} C_VEL
LIN {X 0,Y 378.563,Z 875.57,A -85,B 0,C 180,E1 16896.698,E2 16896.698} C_VEL
LIN {X 0,Y 378.661,Z 872.208,A -85,B 0,C 180,E1 16896.416,E2 16896.416} C_VEL
LIN {X 0,Y 387.542,Z 827.392,A -85,B 0,C 180,E1 16891.739,E2 16891.739} C_VEL
LIN {X 0,Y 398.403,Z 781.578,A -85,B 0,C 180,E1 16886.951,E2 16886.951} C_VEL
LIN {X 0,Y 401.538,Z 769.502,A -85,B 0,C 180,E1 16885.663,E2 16885.663} C_VEL
LIN {X 0,Y 401.412,Z 762.714,A -85,B 0,C 180,E1 16883.638,E2 16883.638} C_VEL
LIN {X 0,Y 401.204,Z 757.688,A -85,B 0,C 180,E1 16881.457,E2 16881.457} C_VEL
LIN {X 0,Y 401.226,Z 756.738,A -85,B 0,C 180,E1 16880.866,E2 16880.866} C_VEL
LIN {X 0,Y 394.89,Z 770.457,A -85,B 0,C 180,E1 16878.196,E2 16878.196} C_VEL
LIN {X 0,Y 390.101,Z 782.767,A -85,B 0,C 180,E1 16877.573,E2 16877.573} C_VEL
LIN {X 0,Y 388.736,Z 786.382,A -85,B 0,C 180,E1 16877.357,E2 16877.357} C_VEL
LIN {X 0,Y 384.096,Z 798.677,A -85,B 0,C 180,E1 16876.791,E2 16876.791} C_VEL
LIN {X 0,Y 382.074,Z 805.273,A -85,B 0,C 180,E1 16876.383,E2 16876.383} C_VEL
LIN {X 0,Y 367.875,Z 976.615,A -85,B 0,C 180,E1 16871.835,E2 16871.835} C_VEL
LIN {X 0,Y 364.943,Z 1001.103,A -85,B 0,C 180,E1 16870.903,E2 16870.903} C_VEL
LIN {X 0,Y 361.47,Z 1024.488,A -85,B 0,C 180,E1 16869.713,E2 16869.713} C_VEL
LIN {X 0,Y 357.866,Z 1045.875,A -85,B 0,C 180,E1 16868.333,E2 16868.333} C_VEL
LIN {X 0,Y 353.771,Z 1067.672,A -85,B 0,C 180,E1 16866.607,E2 16866.607} C_VEL
LIN {X 0,Y 349.546,Z 1088.538,A -85,B 0,C 180,E1 16864.595,E2 16864.595} C_VEL
LIN {X 0,Y 345.473,Z 1107.756,A -85,B 0,C 180,E1 16862.37,E2 16862.37} C_VEL
LIN {X 0,Y 341.679,Z 1125.214,A -85,B 0,C 180,E1 16859.973,E2 16859.973} C_VEL
LIN {X 0,Y 338.11,Z 1141.66,A -85,B 0,C 180,E1 16857.279,E2 16857.279} C_VEL
LIN {X 0,Y 335.103,Z 1156.14,A -85,B 0,C 180,E1 16854.479,E2 16854.479} C_VEL
LIN {X 0,Y 332.487,Z 1169.858,A -85,B 0,C 180,E1 16851.336,E2 16851.336} C_VEL
LIN {X 0,Y 330.579,Z 1181.511,A -85,B 0,C 180,E1 16848.149,E2 16848.149} C_VEL
LIN {X 0,Y 329.267,Z 1191.596,A -85,B 0,C 180,E1 16844.776,E2 16844.776} C_VEL
LIN {X 0,Y 328.572,Z 1199.721,A -85,B 0,C 180,E1 16841.406,E2 16841.406} C_VEL
LIN {X 0,Y 328.34,Z 1206.102,A -85,B 0,C 180,E1 16838.05,E2 16838.05} C_VEL
LIN {X 0,Y 328.35,Z 1210.486,A -85,B 0,C 180,E1 16834.889,E2 16834.889} C_VEL
LIN {X 0,Y 328.387,Z 1213.601,A -85,B 0,C 180,E1 16831.568,E2 16831.568} C_VEL
LIN {X 0,Y 328.306,Z 1215.005,A -85,B 0,C 180,E1 16828.601,E2 16828.601} C_VEL
LIN {X 0,Y 328.116,Z 1215.25,A -85,B 0,C 180,E1 16825.228,E2 16825.228} C_VEL
LIN {X 0,Y 328.085,Z 1213.851,A -85,B 0,C 180,E1 16821.762,E2 16821.762} C_VEL
LIN {X 0,Y 328.586,Z 1210.633,A -85,B 0,C 180,E1 16817.877,E2 16817.877} C_VEL
LIN {X 0,Y 329.901,Z 1205.909,A -85,B 0,C 180,E1 16814.168,E2 16814.168} C_VEL
LIN {X 0,Y 332.374,Z 1199.148,A -85,B 0,C 180,E1 16810.308,E2 16810.308} C_VEL
LIN {X 0,Y 336.331,Z 1190.215,A -85,B 0,C 180,E1 16806.336,E2 16806.336} C_VEL
LIN {X 0,Y 341.559,Z 1179.844,A -85,B 0,C 180,E1 16802.636,E2 16802.636} C_VEL
LIN {X 0,Y 348.583,Z 1166.951,A -85,B 0,C 180,E1 16798.912,E2 16798.912} C_VEL
LIN {X 0,Y 356.854,Z 1152.672,A -85,B 0,C 180,E1 16795.527,E2 16795.527} C_VEL
LIN {X 0,Y 367.202,Z 1135.742,A -85,B 0,C 180,E1 16792.215,E2 16792.215} C_VEL
LIN {X 0,Y 379.301,Z 1116.743,A -85,B 0,C 180,E1 16789.172,E2 16789.172} C_VEL
LIN {X 0,Y 392.619,Z 1096.591,A -85,B 0,C 180,E1 16786.557,E2 16786.557} C_VEL
LIN {X 0,Y 405.9,Z 1076.956,A -85,B 0,C 180,E1 16784.506,E2 16784.506} C_VEL
LIN {X 0,Y 409.186,Z 1072.033,A -85,B 0,C 180,E1 16784.047,E2 16784.047} C_VEL
LIN {X 0,Y 395.711,Z 1090.794,A -85,B 0,C 180,E1 16781.804,E2 16781.804} C_VEL
LIN {X 0,Y 383.021,Z 1108.441,A -85,B 0,C 180,E1 16779.182,E2 16779.182} C_VEL
LIN {X 0,Y 371.216,Z 1124.948,A -85,B 0,C 180,E1 16776.152,E2 16776.152} C_VEL
LIN {X 0,Y 360.998,Z 1139.359,A -85,B 0,C 180,E1 16772.883,E2 16772.883} C_VEL
LIN {X 0,Y 352.131,Z 1151.959,A -85,B 0,C 180,E1 16769.336,E2 16769.336} C_VEL
LIN {X 0,Y 345.09,Z 1162.11,A -85,B 0,C 180,E1 16765.765,E2 16765.765} C_VEL
LIN {X 0,Y 339.557,Z 1170.284,A -85,B 0,C 180,E1 16762.146,E2 16762.146} C_VEL
LIN {X 0,Y 335.101,Z 1176.901,A -85,B 0,C 180,E1 16758.262,E2 16758.262} C_VEL
LIN {X 0,Y 332.056,Z 1181.49,A -85,B 0,C 180,E1 16754.477,E2 16754.477} C_VEL
LIN {X 0,Y 329.988,Z 1184.561,A -85,B 0,C 180,E1 16750.478,E2 16750.478} C_VEL
LIN {X 0,Y 328.927,Z 1185.819,A -85,B 0,C 180,E1 16746.812,E2 16746.812} C_VEL
LIN {X 0,Y 328.404,Z 1185.4,A -85,B 0,C 180,E1 16743.145,E2 16743.145} C_VEL
LIN {X 0,Y 328.215,Z 1183.443,A -85,B 0,C 180,E1 16739.48,E2 16739.48} C_VEL
LIN {X 0,Y 328.196,Z 1180.259,A -85,B 0,C 180,E1 16736.161,E2 16736.161} C_VEL
LIN {X 0,Y 328.384,Z 1175.273,A -85,B 0,C 180,E1 16732.657,E2 16732.657} C_VEL
LIN {X 0,Y 328.919,Z 1168.623,A -85,B 0,C 180,E1 16729.14,E2 16729.14} C_VEL
LIN {X 0,Y 329.873,Z 1160.579,A -85,B 0,C 180,E1 16725.792,E2 16725.792} C_VEL
LIN {X 0,Y 331.401,Z 1150.61,A -85,B 0,C 180,E1 16722.444,E2 16722.444} C_VEL
LIN {X 0,Y 333.6,Z 1138.615,A -85,B 0,C 180,E1 16719.108,E2 16719.108} C_VEL
LIN {X 0,Y 336.189,Z 1125.938,A -85,B 0,C 180,E1 16716.145,E2 16716.145} C_VEL
LIN {X 0,Y 339.397,Z 1111.034,A -85,B 0,C 180,E1 16713.213,E2 16713.213} C_VEL
LIN {X 0,Y 342.995,Z 1094.574,A -85,B 0,C 180,E1 16710.489,E2 16710.489} C_VEL
LIN {X 0,Y 346.906,Z 1076.585,A -85,B 0,C 180,E1 16707.976,E2 16707.976} C_VEL
LIN {X 0,Y 351.024,Z 1056.938,A -85,B 0,C 180,E1 16705.672,E2 16705.672} C_VEL
LIN {X 0,Y 355.087,Z 1036.237,A -85,B 0,C 180,E1 16703.646,E2 16703.646} C_VEL
LIN {X 0,Y 358.786,Z 1015.894,A -85,B 0,C 180,E1 16701.988,E2 16701.988} C_VEL
LIN {X 0,Y 362.365,Z 993.63,A -85,B 0,C 180,E1 16700.509,E2 16700.509} C_VEL
LIN {X 0,Y 365.432,Z 971.201,A -85,B 0,C 180,E1 16699.321,E2 16699.321} C_VEL
LIN {X 0,Y 368.1,Z 947.469,A -85,B 0,C 180,E1 16698.352,E2 16698.352} C_VEL
LIN {X 0,Y 370.837,Z 915.626,A -85,B 0,C 180,E1 16697.427,E2 16697.427} C_VEL
LIN {X 0,Y 384.48,Z 751.102,A -85,B 0,C 180,E1 16693.156,E2 16693.156} C_VEL
LIN {X 0,Y 368.129,Z 721.496,A -85,B 0,C 180,E1 16690.276,E2 16690.276} C_VEL
